C07276=1045.555,91.090,414.139,170.365,36.249,156.822
C07277=1045.549,90.841,414.159,170.363,36.248,156.822
C07278=1045.543,90.592,414.178,170.362,36.246,156.822
C07279=1045.537,90.343,414.197,170.359,36.245,156.821
C07280=1045.531,90.094,414.216,170.357,36.243,156.821
C07281=1045.524,89.845,414.234,170.356,36.242,156.821
C07282=1045.518,89.596,414.253,170.354,36.240,156.820
C07283=1045.512,89.345,414.272,170.352,36.239,156.820
C07284=1045.505,89.096,414.291,170.351,36.238,156.820
C07285=1045.499,88.847,414.310,170.349,36.236,156.820
C07286=1045.493,88.598,414.329,170.346,36.234,156.819
C07287=1045.487,88.349,414.348,170.345,36.233,156.819
C07288=1045.480,88.099,414.366,170.343,36.232,156.819
C07289=1045.474,87.850,414.385,170.341,36.231,156.819
C07290=1045.467,87.601,414.404,170.340,36.229,156.818
C07291=1045.462,87.352,414.423,170.338,36.228,156.818
C07292=1045.455,87.103,414.441,170.335,36.226,156.818
C07293=1045.449,86.854,414.460,170.334,36.224,156.817
C07294=1045.442,86.604,414.479,170.332,36.223,156.817
C07295=1045.437,86.355,414.498,170.330,36.222,156.817
C07296=1045.430,86.106,414.517,170.329,36.221,156.817
C07297=1045.424,85.857,414.535,170.327,36.219,156.816
C07298=1045.418,85.608,414.554,170.325,36.217,156.816
C07299=1045.412,85.358,414.573,170.323,36.216,156.816
C07300=1045.405,85.109,414.592,170.321,36.214,156.816
C07301=1045.399,84.860,414.610,170.319,36.213,156.815
C07302=1045.393,84.611,414.629,170.318,36.212,156.815
C07303=1045.387,84.361,414.648,170.316,36.211,156.815
C07304=1045.380,84.112,414.667,170.314,36.209,156.815
C07305=1045.374,83.863,414.685,170.313,36.207,156.814
C07306=1045.368,83.614,414.703,170.310,36.206,156.814
C07307=1045.362,83.365,414.722,170.308,36.204,156.814
C07308=1045.356,83.116,414.741,170.307,36.203,156.813
C07309=1045.350,82.866,414.760,170.305,36.202,156.813
C07310=1045.344,82.617,414.778,170.303,36.200,156.813
C07311=1045.337,82.368,414.797,170.302,36.199,156.813
C07312=1045.331,82.118,414.815,170.300,36.197,156.812
C07313=1045.325,81.869,414.834,170.297,36.195,156.812
C07314=1045.319,81.620,414.853,170.296,36.194,156.812
C07315=1045.312,81.371,414.872,170.294,36.193,156.812
C07316=1045.306,81.122,414.890,170.292,36.192,156.811
C07317=1045.300,80.873,414.909,170.291,36.190,156.811
C07318=1045.295,80.623,414.927,170.289,36.188,156.811
C07319=1045.288,80.374,414.946,170.288,36.187,156.811
C07320=1045.282,80.125,414.964,170.285,36.185,156.810
C07321=1045.276,79.876,414.983,170.283,36.184,156.810
C07322=1045.269,79.626,415.001,170.282,36.183,156.810
C07323=1045.264,79.408,415.018,170.280,36.181,156.809
C07324=1045.259,79.189,415.034,170.279,36.180,156.809
C07325=1045.254,78.971,415.050,170.277,36.178,156.809
C07326=1045.248,78.752,415.066,170.275,36.177,156.809
C07327=1045.243,78.533,415.083,170.273,36.176,156.808
C07328=1045.237,78.314,415.099,170.272,36.175,156.808
C07329=1045.231,78.096,415.115,170.270,36.173,156.808
C07330=1045.227,77.877,415.131,170.269,36.172,156.808
C07331=1045.219,77.591,415.152,170.267,36.171,156.807
C07332=1045.212,77.306,415.173,170.265,36.169,156.807
C07333=1045.205,77.019,415.194,170.263,36.168,156.807
C07334=1045.198,76.733,415.215,170.260,36.166,156.807
C07335=1045.192,76.484,415.234,170.259,36.164,156.806
C07336=1045.185,76.235,415.252,170.257,36.163,156.806
C07337=1045.179,75.985,415.270,170.255,36.161,156.806
C07338=1045.173,75.736,415.289,170.254,36.160,156.805
C07339=1045.167,75.487,415.307,170.252,36.159,156.805
C07340=1045.160,75.237,415.325,170.250,36.158,156.805
C07341=1045.154,74.988,415.343,170.248,36.156,156.805
C07342=1045.148,74.739,415.362,170.246,36.154,156.804
C07343=1045.142,74.490,415.380,170.244,36.153,156.804
C07344=1045.135,74.241,415.398,170.243,36.152,156.804
C07345=1045.129,73.992,415.416,170.241,36.151,156.804
C07346=1045.122,73.742,415.434,170.239,36.149,156.803
C07347=1045.117,73.494,415.452,170.238,36.147,156.803
C07348=1045.111,73.244,415.470,170.235,36.146,156.803
C07349=1045.104,72.995,415.489,170.233,36.145,156.803
C07350=1045.098,72.745,415.507,170.232,36.143,156.802
C07351=1045.092,72.496,415.526,170.230,36.142,156.802
C07352=1045.085,72.246,415.544,170.228,36.140,156.802
C07353=1045.080,71.998,415.562,170.227,36.139,156.802
C07354=1045.073,71.748,415.580,170.225,36.137,156.801
C07355=1045.067,71.499,415.598,170.222,36.136,156.801
C07356=1045.060,71.249,415.616,170.221,36.135,156.801
C07357=1045.054,71.001,415.634,170.219,36.134,156.801
C07358=1045.048,70.751,415.652,170.217,36.132,156.800
C07359=1045.042,70.502,415.671,170.216,36.130,156.800
C07360=1045.036,70.252,415.689,170.214,36.129,156.800
C07361=1045.030,70.003,415.706,170.213,36.128,156.800
C07362=1045.024,69.754,415.725,170.210,36.126,156.799
C07363=1045.018,69.504,415.743,170.208,36.125,156.799
C07364=1045.010,69.256,415.761,170.207,36.123,156.799
C07365=1045.004,69.006,415.779,170.205,36.122,156.799
C07366=1044.999,68.757,415.796,170.203,36.121,156.798
C07367=1044.992,68.508,415.815,170.202,36.119,156.798
C07368=1044.986,68.258,415.832,170.200,36.118,156.798
C07369=1044.979,68.009,415.850,170.197,36.116,156.797
C07370=1044.974,67.760,415.868,170.196,36.115,156.797
C07371=1044.967,67.510,415.886,170.194,36.114,156.797
C07372=1044.961,67.261,415.904,170.192,36.112,156.797
C07373=1044.954,67.012,415.922,170.191,36.111,156.796
C07374=1044.949,66.763,415.940,170.189,36.109,156.796
C07375=1044.943,66.513,415.958,170.187,36.108,156.796
C07376=1044.935,66.264,415.976,170.186,36.107,156.796
C07377=1044.930,66.015,415.994,170.183,36.106,156.795
C07378=1044.924,65.765,416.011,170.181,36.104,156.795
C07379=1044.917,65.516,416.029,170.180,36.102,156.795
C07380=1044.910,65.267,416.047,170.178,36.101,156.795
C07381=1044.905,65.018,416.065,170.176,36.100,156.794
C07382=1044.898,64.768,416.082,170.174,36.099,156.794
C07383=1044.892,64.519,416.100,170.173,36.097,156.794
C07384=1044.886,64.270,416.119,170.170,36.095,156.794
C07385=1044.880,64.020,416.136,170.168,36.094,156.793
C07386=1044.873,63.771,416.154,170.167,36.093,156.793
C07387=1044.866,63.522,416.171,170.165,36.092,156.793
C07388=1044.861,63.273,416.189,170.163,36.090,156.793
C07389=1044.854,63.023,416.206,170.162,36.089,156.792
C07390=1044.848,62.773,416.224,170.160,36.088,156.792
C07391=1044.841,62.525,416.242,170.158,36.087,156.792
C07392=1044.835,62.276,416.260,170.156,36.085,156.792
C07393=1044.828,62.026,416.277,170.154,36.084,156.792
C07394=1044.822,61.776,416.295,170.152,36.083,156.791
C07395=1044.814,61.491,416.314,170.150,36.081,156.791
C07396=1044.807,61.204,416.335,170.148,36.080,156.791
C07397=1044.800,60.918,416.355,170.146,36.078,156.791
C07398=1044.792,60.632,416.375,170.144,36.076,156.790
C07399=1044.787,60.383,416.392,170.142,36.075,156.790
C07400=1044.780,60.133,416.410,170.140,36.074,156.790
C07401=1044.773,59.884,416.427,170.138,36.073,156.789
C07402=1044.768,59.635,416.445,170.137,36.071,156.789
C07403=1044.760,59.386,416.463,170.135,36.070,156.789
C07404=1044.754,59.136,416.481,170.133,36.069,156.789
C07405=1044.748,58.887,416.498,170.132,36.067,156.789
C07406=1044.742,58.638,416.516,170.130,36.066,156.788
C07407=1044.735,58.388,416.533,170.128,36.065,156.788
C07408=1044.729,58.139,416.550,170.126,36.063,156.788
C07409=1044.723,57.890,416.568,170.124,36.062,156.788
C07410=1044.716,57.641,416.585,170.122,36.060,156.787
C07411=1044.711,57.391,416.602,170.120,36.059,156.787
C07412=1044.704,57.141,416.619,170.119,36.058,156.787
C07413=1044.698,56.892,416.636,170.117,36.057,156.787
C07414=1044.691,56.643,416.654,170.115,36.055,156.786
C07415=1044.685,56.393,416.672,170.113,36.054,156.786
C07416=1044.679,56.144,416.689,170.111,36.053,156.786
C07417=1044.672,55.895,416.706,170.109,36.052,156.786
C07418=1044.666,55.646,416.723,170.108,36.050,156.785
C07419=1044.660,55.396,416.741,170.106,36.048,156.785
C07420=1044.653,55.147,416.759,170.104,36.047,156.785
C07421=1044.647,54.898,416.776,170.103,36.046,156.785
C07422=1044.641,54.648,416.794,170.101,36.045,156.784
C07423=1044.634,54.400,416.811,170.098,36.043,156.784
C07424=1044.628,54.149,416.828,170.097,36.042,156.784
C07425=1044.622,53.901,416.845,170.095,36.041,156.784
C07426=1044.615,53.651,416.862,170.093,36.039,156.783
C07427=1044.610,53.402,416.880,170.091,36.038,156.783
C07428=1044.603,53.153,416.897,170.090,36.037,156.783
C07429=1044.596,52.903,416.914,170.088,36.035,156.783
C07430=1044.591,52.654,416.932,170.086,36.034,156.782
C07431=1044.584,52.404,416.949,170.084,36.032,156.782
C07432=1044.579,52.155,416.966,170.082,36.031,156.782
C07433=1044.572,51.906,416.983,170.080,36.030,156.782
C07434=1044.565,51.657,417.000,170.079,36.029,156.782
C07435=1044.559,51.407,417.018,170.077,36.027,156.781
C07436=1044.553,51.158,417.035,170.075,36.026,156.781
C07437=1044.546,50.908,417.052,170.074,36.024,156.781
C07438=1044.541,50.659,417.070,170.072,36.023,156.780
C07439=1044.534,50.410,417.087,170.069,36.022,156.780
C07440=1044.528,50.161,417.103,170.068,36.020,156.780
C07441=1044.522,49.911,417.121,170.066,36.019,156.780
C07442=1044.516,49.662,417.138,170.064,36.018,156.780
C07443=1044.509,49.413,417.155,170.063,36.016,156.779
C07444=1044.504,49.163,417.172,170.061,36.015,156.779
C07445=1044.497,48.914,417.190,170.059,36.013,156.779
C07446=1044.491,48.665,417.207,170.057,36.012,156.779
C07447=1044.485,48.416,417.224,170.055,36.011,156.778
C07448=1044.479,48.166,417.241,170.053,36.009,156.778
C07449=1044.472,47.917,417.258,170.051,36.008,156.778
C07450=1044.466,47.667,417.276,170.050,36.007,156.778
C07451=1044.460,47.418,417.292,170.048,36.006,156.777
C07452=1044.453,47.169,417.309,170.046,36.004,156.777
C07453=1044.448,46.920,417.327,170.045,36.002,156.777
C07454=1044.441,46.670,417.343,170.043,36.001,156.777
C07455=1044.435,46.421,417.360,170.040,36.000,156.776
C07456=1044.429,46.172,417.378,170.039,35.999,156.776
C07457=1044.423,45.922,417.395,170.037,35.997,156.776
C07458=1044.417,45.673,417.412,170.035,35.996,156.776
C07459=1044.410,45.386,417.431,170.033,35.994,156.775
C07460=1044.402,45.100,417.451,170.031,35.993,156.775
C07461=1044.396,44.813,417.470,170.029,35.991,156.775
C07462=1044.389,44.527,417.490,170.027,35.990,156.775
C07463=1044.382,44.277,417.507,170.025,35.988,156.774
C07464=1044.376,44.029,417.524,170.023,35.986,156.774
C07465=1044.371,43.779,417.541,170.021,35.985,156.774
C07466=1044.364,43.529,417.558,170.020,35.984,156.774
C07467=1044.358,43.280,417.574,170.018,35.983,156.773
C07468=1044.351,43.031,417.592,170.016,35.981,156.773
C07469=1044.345,42.781,417.608,170.015,35.980,156.773
C07470=1044.340,42.532,417.625,170.013,35.979,156.773
C07471=1044.333,42.282,417.642,170.010,35.977,156.772
C07472=1044.327,42.033,417.659,170.009,35.976,156.772
C07473=1044.320,41.783,417.676,170.007,35.975,156.772
C07474=1044.314,41.535,417.693,170.005,35.974,156.772
C07475=1044.308,41.285,417.709,170.003,35.972,156.771
C07476=1044.301,41.036,417.726,170.002,35.971,156.771
C07477=1044.295,40.787,417.743,170.000,35.970,156.771
C07478=1044.289,40.536,417.759,169.998,35.968,156.771
C07479=1044.283,40.288,417.776,169.996,35.967,156.770
C07480=1044.277,40.038,417.792,169.994,35.965,156.770
C07481=1044.270,39.789,417.810,169.992,35.964,156.770
C07482=1044.264,39.540,417.826,169.990,35.963,156.770
C07483=1044.258,39.290,417.842,169.989,35.961,156.770
C07484=1044.251,39.041,417.860,169.987,35.960,156.769
C07485=1044.245,38.792,417.876,169.985,35.959,156.769
C07486=1044.239,38.543,417.893,169.984,35.958,156.769
C07487=1044.232,38.293,417.909,169.981,35.956,156.769
C07488=1044.227,38.043,417.926,169.979,35.955,156.768
C07489=1044.221,37.794,417.943,169.977,35.954,156.768
C07490=1044.214,37.544,417.960,169.976,35.952,156.768
C07491=1044.207,37.295,417.976,169.974,35.951,156.768
C07492=1044.202,37.046,417.992,169.972,35.950,156.767
C07493=1044.195,36.796,418.009,169.970,35.949,156.767
C07494=1044.189,36.547,418.025,169.969,35.947,156.767
C07495=1044.183,36.298,418.042,169.967,35.946,156.767
C07496=1044.176,36.048,418.059,169.964,35.945,156.767
C07497=1044.170,35.799,418.075,169.962,35.943,156.766
C07498=1044.163,35.550,418.091,169.961,35.942,156.766
C07499=1044.157,35.300,418.107,169.959,35.942,156.766
C07500=1044.151,35.051,418.124,169.957,35.940,156.766
C07501=1044.144,34.802,418.141,169.956,35.939,156.766
C07502=1044.138,34.552,418.157,169.954,35.938,156.765
C07503=1044.132,34.302,418.174,169.952,35.936,156.765
C07504=1044.125,34.053,418.189,169.950,35.935,156.765
C07505=1044.119,33.803,418.206,169.948,35.934,156.765
C07506=1044.112,33.555,418.223,169.946,35.933,156.764
C07507=1044.107,33.305,418.239,169.944,35.931,156.764
C07508=1044.101,33.056,418.255,169.942,35.930,156.764
C07509=1044.093,32.806,418.271,169.941,35.929,156.764
C07510=1044.087,32.557,418.288,169.939,35.927,156.763
C07511=1044.081,32.308,418.304,169.937,35.926,156.763
C07512=1044.075,32.059,418.321,169.935,35.925,156.763
C07513=1044.069,31.809,418.338,169.934,35.924,156.763
C07514=1044.062,31.560,418.353,169.931,35.922,156.763
C07515=1044.056,31.310,418.369,169.929,35.921,156.762
C07516=1044.050,31.061,418.386,169.927,35.920,156.762
C07517=1044.043,30.811,418.402,169.926,35.918,156.762
C07518=1044.037,30.562,418.419,169.924,35.917,156.762
C07519=1044.031,30.313,418.434,169.922,35.916,156.761
C07520=1044.025,30.063,418.450,169.920,35.914,156.761
C07521=1044.018,29.813,418.467,169.919,35.914,156.761
C07522=1044.012,29.564,418.484,169.917,35.913,156.761
C07523=1044.005,29.278,418.502,169.914,35.911,156.761
C07524=1043.998,28.991,418.521,169.912,35.909,156.760
C07525=1043.991,28.705,418.540,169.910,35.908,156.760
C07526=1043.984,28.418,418.558,169.908,35.907,156.760
C07527=1043.978,28.169,418.574,169.906,35.905,156.760
C07528=1043.971,27.919,418.590,169.904,35.904,156.759
C07529=1043.965,27.669,418.606,169.903,35.903,156.759
C07530=1043.958,27.420,418.622,169.901,35.902,156.759
C07531=1043.952,27.171,418.638,169.899,35.900,156.759
C07532=1043.946,26.922,418.655,169.896,35.899,156.759
C07533=1043.939,26.672,418.671,169.895,35.898,156.758
C07534=1043.933,26.423,418.687,169.893,35.896,156.758
C07535=1043.927,26.173,418.703,169.891,35.896,156.758
C07536=1043.920,25.924,418.719,169.889,35.894,156.758
C07537=1043.914,25.675,418.735,169.887,35.893,156.757
C07538=1043.907,25.425,418.751,169.886,35.892,156.757
C07539=1043.901,25.176,418.767,169.884,35.891,156.757
C07540=1043.894,24.927,418.783,169.882,35.889,156.757
C07541=1043.889,24.677,418.798,169.879,35.888,156.757
C07542=1043.883,24.427,418.815,169.878,35.887,156.756
C07543=1043.876,24.178,418.830,169.876,35.886,156.756
C07544=1043.869,23.928,418.847,169.874,35.885,156.756
C07545=1043.863,23.679,418.863,169.872,35.883,156.756
C07546=1043.857,23.430,418.879,169.870,35.882,156.756
C07547=1043.850,23.181,418.895,169.869,35.881,156.755
C07548=1043.844,22.931,418.910,169.867,35.880,156.755
C07549=1043.839,22.682,418.926,169.865,35.879,156.755
C07550=1043.832,22.433,418.942,169.863,35.878,156.755
C07551=1043.825,22.183,418.959,169.861,35.876,156.755
C07552=1043.819,21.934,418.974,169.859,35.875,156.754
C07553=1043.813,21.684,418.990,169.857,35.874,156.754
C07554=1043.806,21.434,419.006,169.855,35.872,156.754
C07555=1043.800,21.185,419.022,169.853,35.871,156.754
C07556=1043.794,20.936,419.037,169.852,35.870,156.753
C07557=1043.788,20.686,419.053,169.850,35.869,156.753
C07558=1043.781,20.437,419.069,169.848,35.868,156.753
C07559=1043.775,20.188,419.085,169.846,35.867,156.753
C07560=1043.769,19.938,419.101,169.844,35.865,156.753
C07561=1043.762,19.688,419.116,169.842,35.864,156.752
C07562=1043.756,19.439,419.132,169.840,35.863,156.752
C07563=1043.750,19.190,419.148,169.838,35.861,156.752
C07564=1043.743,18.940,419.163,169.836,35.861,156.752
C07565=1043.737,18.691,419.180,169.834,35.859,156.752
C07566=1043.731,18.442,419.195,169.833,35.858,156.751
C07567=1043.724,18.192,419.210,169.831,35.857,156.751
C07568=1043.718,17.943,419.226,169.829,35.856,156.751
C07569=1043.712,17.694,419.242,169.827,35.855,156.751
C07570=1043.706,17.444,419.258,169.825,35.854,156.751
C07571=1043.699,17.195,419.273,169.823,35.852,156.750
C07572=1043.693,16.946,419.289,169.821,35.851,156.750
C07573=1043.687,16.696,419.305,169.819,35.850,156.750
C07574=1043.680,16.447,419.320,169.817,35.849,156.750
C07575=1043.675,16.197,419.336,169.815,35.848,156.750
C07576=1043.668,15.948,419.351,169.814,35.847,156.749
C07577=1043.661,15.698,419.367,169.812,35.845,156.749
C07578=1043.655,15.448,419.383,169.810,35.844,156.749
C07579=1043.648,15.199,419.399,169.808,35.843,156.749
C07580=1043.643,14.949,419.414,169.806,35.842,156.749
C07581=1043.636,14.700,419.430,169.804,35.841,156.748
C07582=1043.630,14.450,419.445,169.802,35.839,156.748
C07583=1043.624,14.201,419.461,169.800,35.838,156.748
C07584=1043.617,13.951,419.476,169.798,35.837,156.748
C07585=1043.611,13.702,419.492,169.796,35.836,156.748
C07586=1043.604,13.452,419.507,169.794,35.835,156.747
C07587=1043.597,13.167,419.524,169.792,35.834,156.747
C07588=1043.589,12.882,419.542,169.790,35.832,156.747
C07589=1043.582,12.597,419.559,169.788,35.831,156.747
C07590=1043.575,12.312,419.578,169.786,35.830,156.747
C07591=1043.569,12.062,419.592,169.784,35.829,156.746
C07592=1043.562,11.813,419.608,169.781,35.828,156.746
C07593=1043.556,11.564,419.623,169.779,35.827,156.746
C07594=1043.550,11.314,419.638,169.778,35.826,156.746
C07595=1043.543,11.065,419.654,169.776,35.824,156.746
C07596=1043.537,10.815,419.669,169.774,35.823,156.745
C07597=1043.531,10.566,419.685,169.772,35.822,156.745
C07598=1043.524,10.316,419.700,169.770,35.821,156.745
C07599=1043.518,10.067,419.715,169.768,35.820,156.745
C07600=1043.511,9.818,419.730,169.766,35.819,156.745
C07601=1043.505,9.568,419.745,169.765,35.818,156.745
C07602=1043.498,9.318,419.760,169.762,35.817,156.744
C07603=1043.492,9.069,419.776,169.760,35.816,156.744
C07604=1043.485,8.820,419.791,169.758,35.815,156.744
C07605=1043.480,8.570,419.806,169.756,35.813,156.744
C07606=1043.473,8.321,419.822,169.754,35.813,156.744
C07607=1043.467,8.071,419.837,169.752,35.811,156.743
C07608=1043.460,7.821,419.852,169.751,35.810,156.743
C07609=1043.453,7.572,419.868,169.749,35.809,156.743
C07610=1043.447,7.323,419.883,169.747,35.808,156.743
C07611=1043.441,7.073,419.898,169.745,35.807,156.743
C07612=1043.435,6.824,419.912,169.743,35.806,156.743
C07613=1043.428,6.575,419.928,169.741,35.805,156.742
C07614=1043.422,6.325,419.943,169.738,35.803,156.742
C07615=1043.416,6.075,419.958,169.737,35.803,156.742
C07616=1043.410,5.826,419.973,169.735,35.801,156.742
C07617=1043.403,5.577,419.989,169.733,35.800,156.742
C07618=1043.397,5.327,420.004,169.731,35.799,156.741
C07619=1043.390,5.077,420.019,169.729,35.798,156.741
C07620=1043.384,4.828,420.034,169.727,35.797,156.741
C07621=1043.378,4.579,420.048,169.725,35.796,156.741
C07622=1043.372,4.330,420.064,169.724,35.795,156.741
C07623=1043.365,4.080,420.079,169.722,35.794,156.740
C07624=1043.359,3.830,420.094,169.720,35.792,156.740
C07625=1043.352,3.581,420.109,169.717,35.792,156.740
C07626=1043.347,3.331,420.124,169.715,35.790,156.740
C07627=1043.340,3.081,420.139,169.713,35.789,156.740
C07628=1043.334,2.833,420.155,169.711,35.788,156.740
C07629=1043.328,2.583,420.170,169.709,35.787,156.739
C07630=1043.322,2.333,420.185,169.708,35.786,156.739
C07631=1043.315,2.084,420.199,169.706,35.785,156.739
C07632=1043.309,1.834,420.214,169.704,35.784,156.739
C07633=1043.303,1.585,420.229,169.702,35.783,156.739
C07634=1043.297,1.335,420.244,169.700,35.781,156.738
C07635=1043.290,1.086,420.259,169.698,35.781,156.738
C07636=1043.284,0.837,420.275,169.695,35.779,156.738
C07637=1043.277,0.587,420.290,169.693,35.778,156.738
C07638=1043.271,0.338,420.304,169.692,35.777,156.738
C07639=1043.265,0.088,420.319,169.690,35.776,156.737
C07640=1043.259,-0.161,420.334,169.688,35.775,156.737
C07641=1043.252,-0.411,420.349,169.686,35.774,156.737
C07642=1043.246,-0.661,420.364,169.684,35.773,156.737
C07643=1043.241,-0.910,420.379,169.682,35.771,156.737
C07644=1043.234,-1.159,420.394,169.680,35.771,156.737
C07645=1043.228,-1.409,420.409,169.678,35.769,156.736
C07646=1043.222,-1.659,420.424,169.677,35.768,156.736
C07647=1043.216,-1.908,420.438,169.675,35.767,156.736
C07648=1043.209,-2.157,420.453,169.672,35.766,156.736
C07649=1043.203,-2.407,420.468,169.670,35.765,156.736
C07650=1043.197,-2.656,420.483,169.668,35.763,156.735
C07651=1043.190,-2.939,420.499,169.666,35.762,156.735
C07652=1043.182,-3.223,420.517,169.664,35.762,156.735
C07653=1043.176,-3.507,420.534,169.662,35.760,156.735
C07654=1043.169,-3.790,420.550,169.659,35.759,156.735
C07655=1043.162,-4.040,420.564,169.657,35.758,156.734
C07656=1043.156,-4.289,420.579,169.655,35.757,156.734
C07657=1043.150,-4.538,420.594,169.654,35.756,156.734
C07658=1043.143,-4.788,420.609,169.652,35.755,156.734
C07659=1043.136,-5.037,420.623,169.649,35.754,156.734
C07660=1043.130,-5.286,420.638,169.647,35.753,156.734
C07661=1043.124,-5.536,420.652,169.645,35.752,156.733
C07662=1043.118,-5.786,420.667,169.643,35.751,156.733
C07663=1043.111,-6.035,420.681,169.641,35.750,156.733
C07664=1043.105,-6.284,420.696,169.639,35.749,156.733
C07665=1043.098,-6.534,420.711,169.637,35.748,156.733
C07666=1043.092,-6.784,420.724,169.635,35.747,156.733
C07667=1043.086,-7.033,420.739,169.633,35.746,156.732
C07668=1043.080,-7.283,420.754,169.631,35.745,156.732
C07669=1043.073,-7.532,420.769,169.629,35.744,156.732
C07670=1043.066,-7.782,420.783,169.627,35.743,156.732
C07671=1043.061,-8.031,420.797,169.625,35.742,156.732
C07672=1043.054,-8.281,420.812,169.623,35.741,156.732
C07673=1043.047,-8.530,420.826,169.620,35.740,156.731
C07674=1043.042,-8.780,420.840,169.619,35.739,156.731
C07675=1043.035,-9.029,420.855,169.617,35.738,156.731
C07676=1043.028,-9.279,420.870,169.615,35.737,156.731
C07677=1043.022,-9.528,420.884,169.613,35.736,156.731
C07678=1043.016,-9.778,420.898,169.611,35.735,156.731
C07679=1043.010,-10.028,420.913,169.609,35.734,156.730
C07680=1043.003,-10.276,420.927,169.607,35.733,156.730
C07681=1042.997,-10.527,420.942,169.605,35.732,156.730
C07682=1042.991,-10.776,420.956,169.603,35.731,156.730
C07683=1042.984,-11.025,420.971,169.601,35.730,156.730
C07684=1042.978,-11.275,420.985,169.599,35.729,156.730
C07685=1042.972,-11.524,420.999,169.597,35.728,156.729
C07686=1042.965,-11.774,421.014,169.594,35.727,156.729
C07687=1042.959,-12.024,421.028,169.592,35.726,156.729
C07688=1042.953,-12.273,421.042,169.590,35.725,156.729
C07689=1042.947,-12.523,421.056,169.588,35.724,156.729
C07690=1042.941,-12.772,421.071,169.586,35.723,156.729
C07691=1042.934,-13.021,421.086,169.584,35.722,156.728
C07692=1042.928,-13.271,421.099,169.582,35.721,156.728
C07693=1042.922,-13.520,421.114,169.580,35.720,156.728
C07694=1042.916,-13.771,421.128,169.578,35.719,156.728
C07695=1042.909,-14.019,421.142,169.576,35.718,156.728
C07696=1042.903,-14.269,421.157,169.574,35.717,156.728
C07697=1042.897,-14.518,421.171,169.573,35.716,156.728
C07698=1042.890,-14.768,421.185,169.571,35.715,156.727
C07699=1042.885,-15.017,421.199,169.568,35.714,156.727
C07700=1042.878,-15.267,421.214,169.566,35.713,156.727
C07701=1042.872,-15.517,421.228,169.564,35.713,156.727
C07702=1042.865,-15.766,421.242,169.562,35.711,156.727
C07703=1042.859,-16.016,421.256,169.560,35.711,156.727
C07704=1042.853,-16.264,421.270,169.558,35.710,156.727
C07705=1042.846,-16.515,421.284,169.556,35.709,156.726
C07706=1042.840,-16.765,421.298,169.554,35.708,156.726
C07707=1042.834,-17.014,421.312,169.552,35.707,156.726
C07708=1042.827,-17.264,421.326,169.550,35.706,156.726
C07709=1042.820,-17.512,421.340,169.548,35.705,156.726
C07710=1042.814,-17.763,421.354,169.546,35.704,156.726
C07711=1042.808,-18.012,421.367,169.544,35.703,156.725
C07712=1042.802,-18.262,421.382,169.542,35.702,156.725
C07713=1042.796,-18.511,421.396,169.540,35.702,156.725
C07714=1042.789,-18.760,421.411,169.537,35.700,156.725
C07715=1042.782,-19.043,421.426,169.534,35.700,156.725
C07716=1042.775,-19.324,421.442,169.532,35.698,156.725
C07717=1042.768,-19.606,421.458,169.530,35.698,156.725
C07718=1042.761,-19.888,421.473,169.527,35.696,156.724
C07719=1042.754,-20.137,421.487,169.525,35.696,156.724
C07720=1042.748,-20.386,421.501,169.523,35.694,156.724
C07721=1042.742,-20.636,421.515,169.521,35.694,156.724
C07722=1042.735,-20.885,421.529,169.519,35.693,156.724
C07723=1042.729,-21.135,421.543,169.517,35.692,156.724
C07724=1042.723,-21.385,421.556,169.515,35.691,156.724
C07725=1042.717,-21.635,421.570,169.513,35.690,156.723
C07726=1042.710,-21.884,421.584,169.511,35.689,156.723
C07727=1042.703,-22.133,421.598,169.509,35.688,156.723
C07728=1042.698,-22.383,421.612,169.507,35.688,156.723
C07729=1042.691,-22.633,421.626,169.504,35.686,156.723
C07730=1042.684,-22.882,421.640,169.502,35.686,156.723
C07731=1042.678,-23.132,421.654,169.500,35.685,156.723
C07732=1042.672,-23.381,421.667,169.498,35.684,156.722
C07733=1042.667,-23.631,421.681,169.496,35.683,156.722
C07734=1042.660,-23.880,421.695,169.494,35.682,156.722
C07735=1042.653,-24.129,421.709,169.492,35.681,156.722
C07736=1042.647,-24.380,421.723,169.490,35.680,156.722
C07737=1042.641,-24.629,421.736,169.488,35.680,156.722
C07738=1042.635,-24.878,421.749,169.486,35.679,156.722
C07739=1042.628,-25.128,421.764,169.484,35.678,156.721
C07740=1042.622,-25.377,421.778,169.482,35.677,156.721
C07741=1042.615,-25.627,421.791,169.480,35.676,156.721
C07742=1042.610,-25.877,421.805,169.478,35.675,156.721
C07743=1042.604,-26.126,421.818,169.476,35.674,156.721
C07744=1042.598,-26.376,421.833,169.474,35.674,156.721
C07745=1042.591,-26.625,421.846,169.471,35.672,156.721
C07746=1042.585,-26.874,421.860,169.469,35.672,156.720
C07747=1042.578,-27.124,421.873,169.467,35.671,156.720
C07748=1042.573,-27.374,421.887,169.464,35.670,156.720
C07749=1042.566,-27.624,421.901,169.462,35.669,156.720
C07750=1042.560,-27.873,421.914,169.460,35.668,156.720
C07751=1042.553,-28.122,421.927,169.458,35.668,156.720
C07752=1042.547,-28.372,421.941,169.456,35.667,156.720
C07753=1042.540,-28.621,421.954,169.454,35.666,156.720
C07754=1042.534,-28.871,421.968,169.452,35.666,156.720
C07755=1042.527,-29.121,421.981,169.450,35.664,156.719
C07756=1042.522,-29.370,421.995,169.448,35.664,156.719
C07757=1042.515,-29.620,422.009,169.446,35.663,156.719
C07758=1042.509,-29.869,422.022,169.444,35.662,156.719
C07759=1042.503,-30.119,422.035,169.442,35.661,156.719
C07760=1042.496,-30.369,422.049,169.440,35.661,156.719
C07761=1042.490,-30.618,422.062,169.437,35.659,156.719
C07762=1042.483,-30.867,422.075,169.435,35.659,156.718
C07763=1042.477,-31.117,422.089,169.432,35.658,156.718
C07764=1042.470,-31.366,422.102,169.430,35.657,156.718
C07765=1042.464,-31.616,422.115,169.428,35.657,156.718
C07766=1042.458,-31.867,422.129,169.426,35.656,156.718
C07767=1042.452,-32.116,422.142,169.424,35.655,156.718
C07768=1042.446,-32.365,422.156,169.422,35.654,156.718
C07769=1042.439,-32.615,422.169,169.420,35.653,156.718
C07770=1042.433,-32.864,422.183,169.418,35.653,156.718
C07771=1042.427,-33.114,422.196,169.416,35.652,156.717
C07772=1042.420,-33.363,422.209,169.413,35.651,156.717
C07773=1042.414,-33.613,422.223,169.411,35.651,156.717
C07774=1042.408,-33.863,422.235,169.409,35.650,156.717
C07775=1042.402,-34.112,422.249,169.407,35.649,156.717
C07776=1042.395,-34.361,422.262,169.405,35.648,156.717
C07777=1042.389,-34.611,422.276,169.403,35.647,156.717
C07778=1042.382,-34.860,422.289,169.401,35.647,156.717
C07779=1042.376,-35.142,422.304,169.398,35.646,156.716
C07780=1042.369,-35.422,422.319,169.396,35.644,156.716
C07781=1042.362,-35.704,422.334,169.394,35.644,156.716
C07782=1042.354,-35.985,422.349,169.390,35.643,156.716
C07783=1042.348,-36.234,422.362,169.388,35.642,156.716
C07784=1042.342,-36.484,422.375,169.386,35.642,156.716
C07785=1042.336,-36.733,422.388,169.384,35.641,156.716
C07786=1042.330,-36.982,422.401,169.382,35.640,156.716
C07787=1042.323,-37.232,422.415,169.380,35.639,156.715
C07788=1042.317,-37.482,422.427,169.378,35.638,156.715
C07789=1042.311,-37.732,422.441,169.376,35.638,156.715
C07790=1042.305,-37.981,422.454,169.373,35.637,156.715
C07791=1042.299,-38.231,422.466,169.371,35.636,156.715
C07792=1042.292,-38.481,422.480,169.369,35.636,156.715
C07793=1042.286,-38.730,422.493,169.367,35.635,156.715
C07794=1042.280,-38.980,422.506,169.365,35.634,156.715
C07795=1042.274,-39.229,422.519,169.363,35.634,156.715
C07796=1042.267,-39.478,422.532,169.361,35.633,156.715
C07797=1042.261,-39.729,422.545,169.358,35.632,156.714
C07798=1042.255,-39.978,422.559,169.356,35.631,156.714
C07799=1042.248,-40.227,422.571,169.354,35.631,156.714
C07800=1042.242,-40.477,422.584,169.352,35.630,156.714
C07801=1042.236,-40.726,422.597,169.350,35.629,156.714
C07802=1042.229,-40.977,422.610,169.348,35.629,156.714
C07803=1042.223,-41.226,422.623,169.345,35.628,156.714
C07804=1042.216,-41.476,422.635,169.342,35.627,156.714
C07805=1042.210,-41.725,422.648,169.340,35.627,156.714
C07806=1042.204,-41.974,422.662,169.338,35.626,156.714
C07807=1042.198,-42.224,422.674,169.336,35.625,156.713
C07808=1042.192,-42.473,422.688,169.334,35.625,156.713
C07809=1042.184,-42.724,422.700,169.332,35.624,156.713
C07810=1042.178,-42.973,422.713,169.329,35.623,156.713
C07811=1042.172,-43.223,422.726,169.327,35.622,156.713
C07812=1042.166,-43.472,422.739,169.325,35.622,156.713
C07813=1042.160,-43.722,422.752,169.323,35.621,156.713
C07814=1042.153,-43.971,422.764,169.321,35.621,156.713
C07815=1042.147,-44.221,422.777,169.319,35.620,156.713
C07816=1042.141,-44.470,422.790,169.316,35.620,156.713
C07817=1042.135,-44.720,422.803,169.314,35.619,156.713
C07818=1042.128,-44.970,422.816,169.312,35.618,156.712
C07819=1042.122,-45.219,422.828,169.310,35.618,156.712
C07820=1042.116,-45.469,422.841,169.308,35.617,156.712
C07821=1042.110,-45.719,422.854,169.306,35.616,156.712
C07822=1042.104,-45.969,422.867,169.303,35.615,156.712
C07823=1042.097,-46.217,422.879,169.301,35.615,156.712
C07824=1042.091,-46.467,422.892,169.299,35.614,156.712
C07825=1042.085,-46.717,422.904,169.297,35.613,156.712
C07826=1042.079,-46.967,422.918,169.295,35.613,156.712
C07827=1042.072,-47.216,422.930,169.291,35.612,156.711
C07828=1042.066,-47.465,422.943,169.290,35.612,156.712
C07829=1042.060,-47.715,422.955,169.287,35.611,156.711
C07830=1042.054,-47.965,422.968,169.285,35.611,156.711
C07831=1042.047,-48.214,422.981,169.283,35.610,156.711
C07832=1042.041,-48.464,422.993,169.281,35.609,156.711
C07833=1042.035,-48.714,423.006,169.278,35.609,156.711
C07834=1042.029,-48.963,423.019,169.276,35.608,156.711
C07835=1042.022,-49.213,423.031,169.274,35.607,156.711
C07836=1042.016,-49.463,423.044,169.272,35.606,156.711
C07837=1042.010,-49.712,423.057,169.270,35.606,156.711
C07838=1042.004,-49.961,423.069,169.267,35.605,156.710
C07839=1041.998,-50.211,423.081,169.265,35.605,156.711
C07840=1041.992,-50.461,423.094,169.263,35.604,156.710
C07841=1041.985,-50.710,423.107,169.261,35.604,156.710
C07842=1041.979,-50.960,423.119,169.259,35.603,156.710
C07843=1041.972,-51.242,423.133,169.256,35.603,156.710
C07844=1041.964,-51.523,423.147,169.254,35.602,156.710
C07845=1041.957,-51.805,423.160,169.251,35.601,156.710
C07846=1041.950,-52.086,423.174,169.248,35.601,156.710
C07847=1041.943,-52.335,423.186,169.246,35.601,156.710
C07848=1041.937,-52.585,423.199,169.244,35.600,156.710
C07849=1041.931,-52.835,423.211,169.242,35.599,156.710
C07850=1041.925,-53.084,423.224,169.239,35.599,156.710
C07851=1041.918,-53.334,423.236,169.237,35.599,156.710
C07852=1041.911,-53.583,423.248,169.235,35.598,156.710
C07853=1041.905,-53.833,423.261,169.233,35.598,156.710
C07854=1041.899,-54.083,423.273,169.230,35.597,156.709
C07855=1041.892,-54.332,423.285,169.228,35.596,156.709
C07856=1041.886,-54.582,423.297,169.226,35.596,156.709
C07857=1041.880,-54.832,423.309,169.224,35.596,156.709
C07858=1041.874,-55.082,423.322,169.221,35.596,156.709
C07859=1041.867,-55.331,423.334,169.219,35.595,156.709
C07860=1041.860,-55.581,423.346,169.216,35.594,156.709
C07861=1041.854,-55.831,423.358,169.214,35.594,156.709
C07862=1041.848,-56.080,423.370,169.211,35.593,156.709
C07863=1041.841,-56.330,423.382,169.209,35.593,156.709
C07864=1041.835,-56.580,423.395,169.207,35.593,156.709
C07865=1041.829,-56.829,423.407,169.205,35.592,156.709
C07866=1041.823,-57.078,423.418,169.202,35.592,156.709
C07867=1041.817,-57.328,423.431,169.200,35.591,156.709
C07868=1041.810,-57.578,423.443,169.198,35.591,156.709
C07869=1041.804,-57.828,423.455,169.196,35.591,156.709
C07870=1041.797,-58.077,423.467,169.193,35.590,156.709
C07871=1041.791,-58.327,423.479,169.191,35.589,156.708
C07872=1041.785,-58.577,423.492,169.189,35.589,156.708
C07873=1041.778,-58.826,423.504,169.187,35.588,156.708
C07874=1041.772,-59.075,423.515,169.184,35.588,156.708
C07875=1041.766,-59.325,423.528,169.182,35.588,156.708
C07876=1041.760,-59.574,423.540,169.180,35.587,156.708
C07877=1041.753,-59.824,423.552,169.177,35.587,156.708
C07878=1041.747,-60.074,423.564,169.175,35.586,156.708
C07879=1041.740,-60.323,423.576,169.173,35.586,156.708
C07880=1041.734,-60.574,423.587,169.171,35.585,156.708
C07881=1041.729,-60.823,423.600,169.168,35.585,156.708
C07882=1041.722,-61.072,423.612,169.166,35.585,156.708
C07883=1041.715,-61.322,423.624,169.164,35.584,156.708
C07884=1041.710,-61.572,423.636,169.161,35.584,156.708
C07885=1041.703,-61.821,423.648,169.159,35.583,156.708
C07886=1041.697,-62.070,423.660,169.157,35.583,156.708
C07887=1041.691,-62.321,423.671,169.155,35.582,156.708
C07888=1041.685,-62.570,423.683,169.152,35.582,156.708
C07889=1041.678,-62.820,423.695,169.150,35.582,156.708
C07890=1041.671,-63.070,423.707,169.148,35.581,156.707
C07891=1041.666,-63.319,423.720,169.146,35.581,156.707
C07892=1041.660,-63.569,423.731,169.143,35.580,156.707
C07893=1041.653,-63.818,423.743,169.141,35.580,156.707
C07894=1041.647,-64.068,423.755,169.139,35.579,156.707
C07895=1041.641,-64.317,423.767,169.136,35.579,156.707
C07896=1041.635,-64.567,423.778,169.134,35.579,156.707
C07897=1041.628,-64.817,423.790,169.132,35.578,156.707
C07898=1041.622,-65.067,423.803,169.129,35.578,156.707
C07899=1041.616,-65.316,423.814,169.127,35.577,156.707
C07900=1041.610,-65.566,423.826,169.125,35.577,156.707
C07901=1041.604,-65.816,423.838,169.123,35.577,156.707
C07902=1041.598,-66.065,423.850,169.120,35.576,156.707
C07903=1041.592,-66.315,423.861,169.118,35.576,156.707
C07904=1041.585,-66.564,423.873,169.116,35.576,156.707
C07905=1041.580,-66.814,423.885,169.113,35.575,156.707
C07906=1041.573,-67.064,423.896,169.111,35.575,156.707
C07907=1041.566,-67.346,423.910,169.108,35.574,156.707
C07908=1041.559,-67.629,423.923,169.105,35.574,156.707
C07909=1041.552,-67.912,423.936,169.103,35.573,156.707
C07910=1041.545,-68.195,423.949,169.100,35.573,156.706
C07911=1041.539,-68.444,423.961,169.097,35.573,156.707
C07912=1041.533,-68.693,423.974,169.095,35.572,156.706
C07913=1041.527,-68.944,423.985,169.093,35.572,156.706
C07914=1041.520,-69.193,423.997,169.090,35.571,156.706
C07915=1041.515,-69.443,424.008,169.088,35.571,156.706
C07916=1041.509,-69.693,424.020,169.086,35.570,156.706
C07917=1041.502,-69.942,424.032,169.084,35.570,156.706
C07918=1041.496,-70.192,424.043,169.081,35.570,156.706
C07919=1041.490,-70.441,424.055,169.079,35.570,156.706
C07920=1041.485,-70.691,424.066,169.077,35.569,156.706
C07921=1041.478,-70.941,424.078,169.074,35.569,156.706
C07922=1041.472,-71.191,424.090,169.072,35.568,156.706
C07923=1041.466,-71.440,424.101,169.070,35.568,156.706
C07924=1041.460,-71.690,424.113,169.067,35.567,156.706
C07925=1041.454,-71.939,424.125,169.065,35.567,156.706
C07926=1041.448,-72.189,424.136,169.063,35.567,156.706
C07927=1041.441,-72.439,424.148,169.060,35.567,156.706
C07928=1041.435,-72.688,424.159,169.058,35.566,156.706
C07929=1041.429,-72.938,424.171,169.056,35.566,156.706
C07930=1041.424,-73.188,424.182,169.053,35.565,156.706
C07931=1041.417,-73.437,424.194,169.051,35.565,156.706
C07932=1041.411,-73.687,424.205,169.049,35.564,156.706
C07933=1041.406,-73.937,424.217,169.046,35.564,156.706
C07934=1041.400,-74.186,424.228,169.044,35.564,156.706
C07935=1041.393,-74.436,424.240,169.042,35.564,156.705
C07936=1041.386,-74.685,424.251,169.039,35.563,156.705
C07937=1041.380,-74.935,424.262,169.037,35.563,156.706
C07938=1041.374,-75.185,424.273,169.035,35.563,156.705
C07939=1041.368,-75.434,424.285,169.032,35.563,156.705
C07940=1041.361,-75.684,424.296,169.030,35.563,156.705
C07941=1041.356,-75.934,424.307,169.028,35.563,156.705
C07942=1041.349,-76.183,424.319,169.025,35.562,156.705
C07943=1041.343,-76.433,424.330,169.023,35.562,156.705
C07944=1041.337,-76.683,424.341,169.020,35.562,156.705
C07945=1041.331,-76.933,424.352,169.018,35.562,156.705
C07946=1041.325,-77.182,424.364,169.016,35.561,156.705
C07947=1041.318,-77.432,424.375,169.013,35.561,156.705
C07948=1041.313,-77.682,424.386,169.011,35.561,156.705
C07949=1041.306,-77.931,424.398,169.009,35.561,156.705
C07950=1041.300,-78.181,424.409,169.006,35.560,156.705
C07951=1041.294,-78.431,424.420,169.004,35.560,156.705
C07952=1041.288,-78.680,424.431,169.002,35.560,156.705
C07953=1041.282,-78.931,424.442,168.999,35.560,156.705
C07954=1041.276,-79.180,424.454,168.997,35.559,156.705
C07955=1041.269,-79.430,424.465,168.994,35.559,156.705
C07956=1041.263,-79.679,424.475,168.992,35.559,156.705
C07957=1041.256,-79.929,424.486,168.990,35.559,156.705
C07958=1041.251,-80.179,424.497,168.987,35.559,156.705
C07959=1041.244,-80.429,424.509,168.985,35.559,156.705
C07960=1041.238,-80.677,424.520,168.982,35.559,156.705
C07961=1041.231,-80.928,424.531,168.980,35.558,156.705
C07962=1041.226,-81.177,424.542,168.978,35.558,156.705
C07963=1041.219,-81.427,424.553,168.975,35.558,156.705
C07964=1041.213,-81.676,424.563,168.973,35.558,156.705
C07965=1041.206,-81.927,424.574,168.970,35.558,156.705
C07966=1041.201,-82.176,424.585,168.968,35.558,156.705
C07967=1041.194,-82.425,424.596,168.966,35.558,156.705
C07968=1041.188,-82.675,424.607,168.963,35.558,156.705
C07969=1041.182,-82.925,424.618,168.961,35.558,156.705
C07970=1041.175,-83.175,424.628,168.958,35.558,156.705
C07971=1041.168,-83.459,424.641,168.956,35.558,156.705
C07972=1041.161,-83.744,424.654,168.953,35.557,156.705
C07973=1041.154,-84.030,424.666,168.950,35.557,156.705
C07974=1041.147,-84.314,424.678,168.947,35.557,156.705
C07975=1041.140,-84.564,424.689,168.945,35.557,156.705
C07976=1041.135,-84.814,424.700,168.942,35.557,156.705
C07977=1041.129,-85.063,424.711,168.940,35.557,156.705
C07978=1041.122,-85.313,424.721,168.938,35.557,156.705
C07979=1041.116,-85.563,424.732,168.935,35.557,156.705
C07980=1041.110,-85.813,424.743,168.933,35.557,156.705
C07981=1041.103,-86.062,424.754,168.930,35.557,156.705
C07982=1041.097,-86.312,424.765,168.928,35.557,156.705
C07983=1041.091,-86.562,424.776,168.925,35.557,156.706
C07984=1041.085,-86.811,424.786,168.923,35.557,156.706
C07985=1041.079,-87.060,424.797,168.921,35.557,156.706
C07986=1041.073,-87.311,424.808,168.918,35.557,156.706
C07987=1041.066,-87.560,424.818,168.916,35.557,156.706
C07988=1041.060,-87.810,424.830,168.913,35.556,156.706
C07989=1041.053,-88.059,424.840,168.911,35.556,156.706
C07990=1041.048,-88.309,424.850,168.908,35.556,156.706
C07991=1041.042,-88.559,424.861,168.906,35.556,156.706
C07992=1041.035,-88.809,424.872,168.904,35.556,156.706
C07993=1041.029,-89.058,424.883,168.901,35.556,156.706
C07994=1041.023,-89.308,424.893,168.899,35.556,156.706
C07995=1041.016,-89.557,424.904,168.896,35.556,156.706
C07996=1041.011,-89.808,424.914,168.894,35.556,156.706
C07997=1041.005,-90.057,424.925,168.891,35.556,156.706
C07998=1040.998,-90.307,424.936,168.889,35.556,156.706
C07999=1040.992,-90.556,424.947,168.886,35.556,156.706
C08000=1040.986,-90.806,424.957,168.884,35.556,156.706
C08001=1040.981,-91.056,424.967,168.882,35.556,156.706
C08002=1040.974,-91.306,424.978,168.879,35.556,156.706
C08003=1040.968,-91.555,424.989,168.877,35.556,156.706
C08004=1040.962,-91.805,424.999,168.874,35.556,156.706
C08005=1040.956,-92.054,425.009,168.872,35.556,156.706
C08006=1040.949,-92.305,425.020,168.869,35.556,156.706
C08007=1040.944,-92.554,425.031,168.868,35.556,156.706
C08008=1040.937,-92.803,425.041,168.865,35.556,156.706
C08009=1040.932,-93.053,425.052,168.863,35.556,156.706
C08010=1040.925,-93.303,425.062,168.861,35.556,156.706
C08011=1040.919,-93.553,425.073,168.858,35.556,156.706
C08012=1040.914,-93.803,425.083,168.856,35.556,156.706
C08013=1040.907,-94.052,425.094,168.853,35.556,156.706
C08014=1040.901,-94.302,425.104,168.851,35.556,156.706
C08015=1040.895,-94.552,425.114,168.848,35.556,156.706
C08016=1040.889,-94.802,425.125,168.846,35.556,156.706
C08017=1040.882,-95.051,425.136,168.843,35.556,156.706
C08018=1040.877,-95.301,425.146,168.841,35.556,156.706
C08019=1040.871,-95.550,425.157,168.839,35.556,156.706
C08020=1040.865,-95.799,425.167,168.836,35.556,156.706
C08021=1040.859,-96.050,425.177,168.834,35.556,156.706
C08022=1040.852,-96.299,425.188,168.831,35.556,156.706
C08023=1040.847,-96.550,425.198,168.829,35.556,156.706
C08024=1040.840,-96.799,425.208,168.826,35.556,156.706
C08025=1040.835,-97.048,425.219,168.824,35.556,156.706
C08026=1040.829,-97.298,425.229,168.821,35.556,156.706
C08027=1040.823,-97.548,425.239,168.819,35.557,156.707
C08028=1040.816,-97.798,425.249,168.816,35.557,156.707
C08029=1040.810,-98.048,425.260,168.814,35.557,156.707
C08030=1040.804,-98.297,425.270,168.811,35.556,156.707
C08031=1040.797,-98.546,425.280,168.809,35.557,156.707
C08032=1040.792,-98.797,425.290,168.806,35.557,156.707
C08033=1040.786,-99.046,425.301,168.804,35.557,156.707
C08034=1040.779,-99.296,425.310,168.801,35.558,156.707
C08035=1040.773,-99.583,425.322,168.799,35.557,156.707
C08036=1040.765,-99.870,425.334,168.796,35.558,156.707
C08037=1040.758,-100.157,425.345,168.793,35.558,156.707
C08038=1040.751,-100.445,425.357,168.790,35.558,156.707
C08039=1040.745,-100.694,425.367,168.787,35.558,156.707
C08040=1040.739,-100.944,425.377,168.785,35.558,156.707
C08041=1040.733,-101.194,425.387,168.782,35.558,156.707
C08042=1040.727,-101.443,425.397,168.780,35.559,156.707
C08043=1040.720,-101.694,425.407,168.777,35.559,156.707
C08044=1040.714,-101.943,425.418,168.775,35.559,156.708
C08045=1040.708,-102.193,425.428,168.772,35.559,156.708
C08046=1040.702,-102.443,425.437,168.770,35.559,156.708
C08047=1040.696,-102.692,425.448,168.767,35.560,156.708
C08048=1040.690,-102.942,425.458,168.765,35.560,156.708
C08049=1040.684,-103.192,425.467,168.762,35.560,156.708
C08050=1040.677,-103.441,425.477,168.760,35.560,156.708
C08051=1040.672,-103.691,425.488,168.757,35.560,156.708
C08052=1040.666,-103.941,425.497,168.756,35.561,156.708
C08053=1040.660,-104.191,425.507,168.753,35.561,156.708
C08054=1040.653,-104.440,425.517,168.751,35.561,156.708
C08055=1040.648,-104.690,425.527,168.748,35.561,156.708
C08056=1040.641,-104.940,425.537,168.746,35.561,156.708
C08057=1040.635,-105.189,425.547,168.743,35.562,156.708
C08058=1040.629,-105.439,425.557,168.741,35.562,156.708
C08059=1040.623,-105.689,425.567,168.738,35.562,156.708
C08060=1040.617,-105.939,425.576,168.736,35.562,156.708
C08061=1040.611,-106.188,425.587,168.733,35.563,156.709
C08062=1040.605,-106.438,425.596,168.731,35.563,156.709
C08063=1040.599,-106.688,425.606,168.728,35.563,156.709
C08064=1040.593,-106.938,425.616,168.726,35.563,156.709
C08065=1040.587,-107.187,425.626,168.723,35.564,156.709
C08066=1040.581,-107.437,425.635,168.721,35.564,156.709
C08067=1040.574,-107.686,425.645,168.718,35.565,156.709
C08068=1040.568,-107.936,425.655,168.716,35.564,156.709
C08069=1040.562,-108.186,425.665,168.713,35.565,156.709
C08070=1040.556,-108.436,425.675,168.711,35.565,156.709
C08071=1040.550,-108.686,425.684,168.708,35.566,156.709
C08072=1040.544,-108.936,425.694,168.706,35.566,156.709
C08073=1040.538,-109.185,425.703,168.703,35.566,156.709
C08074=1040.532,-109.435,425.713,168.701,35.567,156.710
C08075=1040.525,-109.684,425.723,168.698,35.567,156.710
C08076=1040.519,-109.934,425.733,168.695,35.567,156.710
C08077=1040.513,-110.184,425.742,168.693,35.567,156.710
C08078=1040.507,-110.434,425.752,168.690,35.568,156.710
C08079=1040.501,-110.684,425.761,168.688,35.568,156.710
C08080=1040.495,-110.933,425.771,168.685,35.568,156.710
C08081=1040.489,-111.182,425.780,168.684,35.569,156.710
C08082=1040.483,-111.432,425.790,168.681,35.569,156.710
C08083=1040.476,-111.682,425.799,168.679,35.569,156.710
C08084=1040.471,-111.932,425.810,168.676,35.570,156.710
C08085=1040.465,-112.182,425.819,168.674,35.570,156.710
C08086=1040.459,-112.432,425.829,168.671,35.570,156.711
C08087=1040.452,-112.682,425.838,168.668,35.571,156.711
C08088=1040.446,-112.931,425.848,168.666,35.571,156.711
C08089=1040.441,-113.180,425.857,168.663,35.572,156.711
C08090=1040.435,-113.430,425.867,168.661,35.572,156.711
C08091=1040.428,-113.680,425.876,168.658,35.572,156.711
C08092=1040.422,-113.930,425.886,168.656,35.573,156.711
C08093=1040.416,-114.180,425.895,168.653,35.573,156.711
C08094=1040.410,-114.430,425.904,168.651,35.573,156.711
C08095=1040.404,-114.680,425.914,168.648,35.574,156.711
C08096=1040.398,-114.929,425.923,168.646,35.574,156.711
C08097=1040.392,-115.179,425.932,168.643,35.575,156.712
C08098=1040.386,-115.429,425.942,168.640,35.575,156.712
C08099=1040.379,-115.715,425.952,168.637,35.576,156.712
C08100=1040.372,-116.001,425.963,168.635,35.576,156.712
C08101=1040.365,-116.287,425.975,168.632,35.577,156.712
C08102=1040.357,-116.574,425.985,168.629,35.577,156.712
C08103=1040.352,-116.823,425.994,168.627,35.578,156.712
C08104=1040.346,-117.073,426.003,168.625,35.578,156.712
C08105=1040.340,-117.323,426.013,168.622,35.578,156.712
C08106=1040.334,-117.573,426.022,168.619,35.579,156.712
C08107=1040.328,-117.823,426.032,168.617,35.580,156.713
C08108=1040.322,-118.072,426.041,168.614,35.580,156.713
C08109=1040.315,-118.322,426.049,168.612,35.580,156.713
C08110=1040.309,-118.572,426.059,168.609,35.581,156.713
C08111=1040.303,-118.821,426.068,168.607,35.581,156.713
C08112=1040.297,-119.071,426.078,168.604,35.582,156.713
C08113=1040.292,-119.321,426.086,168.601,35.582,156.713
C08114=1040.285,-119.571,426.096,168.599,35.583,156.713
C08115=1040.279,-119.821,426.106,168.596,35.583,156.713
C08116=1040.273,-120.070,426.113,168.594,35.584,156.714
C08117=1040.267,-120.320,426.123,168.591,35.584,156.714
C08118=1040.261,-120.570,426.133,168.589,35.585,156.714
C08119=1040.255,-120.819,426.142,168.586,35.585,156.714
C08120=1040.249,-121.069,426.151,168.583,35.586,156.714
C08121=1040.243,-121.319,426.160,168.581,35.587,156.714
C08122=1040.236,-121.568,426.169,168.579,35.587,156.714
C08123=1040.230,-121.819,426.178,168.577,35.587,156.714
C08124=1040.225,-122.068,426.187,168.574,35.588,156.714
C08125=1040.219,-122.318,426.196,168.571,35.588,156.715
C08126=1040.213,-122.568,426.206,168.569,35.589,156.715
C08127=1040.207,-122.817,426.215,168.566,35.589,156.715
C08128=1040.201,-123.067,426.223,168.564,35.590,156.715
C08129=1040.195,-123.317,426.233,168.561,35.591,156.715
C08130=1040.189,-123.567,426.241,168.559,35.591,156.715
C08131=1040.183,-123.817,426.251,168.556,35.592,156.715
C08132=1040.176,-124.066,426.260,168.553,35.592,156.715
C08133=1040.170,-124.316,426.269,168.551,35.593,156.716
C08134=1040.165,-124.566,426.278,168.548,35.594,156.716
C08135=1040.159,-124.816,426.287,168.546,35.594,156.716
C08136=1040.152,-125.065,426.296,168.543,35.595,156.716
C08137=1040.147,-125.315,426.304,168.540,35.595,156.716
C08138=1040.141,-125.565,426.314,168.538,35.596,156.716
C08139=1040.134,-125.815,426.322,168.535,35.597,156.716
C08140=1040.128,-126.064,426.331,168.534,35.597,156.716
C08141=1040.123,-126.315,426.340,168.531,35.598,156.717
C08142=1040.116,-126.563,426.349,168.528,35.598,156.717
C08143=1040.110,-126.814,426.357,168.526,35.599,156.717
C08144=1040.104,-127.064,426.367,168.523,35.599,156.717
C08145=1040.098,-127.313,426.375,168.521,35.600,156.717
C08146=1040.092,-127.563,426.384,168.518,35.601,156.717
C08147=1040.087,-127.813,426.393,168.515,35.601,156.717
C08148=1040.081,-128.062,426.402,168.513,35.602,156.717
C08149=1040.076,-128.312,426.412,168.511,35.602,156.717
C08150=1040.073,-128.562,426.423,168.508,35.601,156.717
C08151=1040.070,-128.812,426.433,168.506,35.600,156.717
C08152=1040.067,-129.061,426.445,168.504,35.598,156.717
C08153=1040.066,-129.312,426.458,168.503,35.596,156.717
C08154=1040.066,-129.561,426.471,168.500,35.594,156.716
C08155=1040.066,-129.812,426.484,168.498,35.591,156.716
C08156=1040.067,-130.061,426.498,168.497,35.587,156.715
C08157=1040.068,-130.312,426.513,168.496,35.584,156.715
C08158=1040.072,-130.562,426.528,168.494,35.579,156.714
C08159=1040.076,-130.812,426.544,168.493,35.575,156.713
C08160=1040.080,-131.063,426.561,168.492,35.569,156.712
C08161=1040.085,-131.313,426.577,168.491,35.563,156.711
C08162=1040.090,-131.562,426.595,168.490,35.558,156.710
C08163=1039.746,-131.587,426.335,168.442,35.755,156.744
C08164=1039.739,-131.337,426.317,168.444,35.761,156.745
C08165=1039.734,-131.087,426.300,168.444,35.766,156.746
C08166=1039.730,-130.837,426.284,168.446,35.772,156.747
C08167=1039.726,-130.586,426.268,168.447,35.777,156.748
C08168=1039.724,-130.336,426.252,168.448,35.781,156.748
C08169=1039.722,-130.087,426.237,168.450,35.785,156.749
C08170=1039.720,-129.835,426.223,168.452,35.788,156.749
C08171=1039.721,-129.585,426.210,168.453,35.791,156.750
C08172=1039.721,-129.336,426.196,168.455,35.793,156.750
C08173=1039.722,-129.086,426.184,168.456,35.795,156.751
C08174=1039.724,-128.836,426.173,168.459,35.797,156.751
C08175=1039.727,-128.586,426.162,168.461,35.798,156.751
C08176=1039.731,-128.336,426.151,168.464,35.799,156.751
C08177=1039.735,-128.086,426.141,168.466,35.799,156.751
C08178=1039.740,-127.837,426.131,168.468,35.799,156.751
C08179=1039.746,-127.588,426.123,168.471,35.798,156.751
C08180=1039.752,-127.338,426.114,168.473,35.798,156.751
C08181=1039.758,-127.087,426.105,168.475,35.797,156.751
C08182=1039.765,-126.839,426.096,168.478,35.796,156.751
C08183=1039.771,-126.588,426.087,168.480,35.795,156.750
C08184=1039.776,-126.338,426.079,168.483,35.795,156.750
C08185=1039.783,-126.089,426.070,168.486,35.794,156.750
C08186=1039.789,-125.839,426.061,168.488,35.793,156.750
C08187=1039.794,-125.589,426.052,168.491,35.793,156.750
C08188=1039.801,-125.339,426.044,168.494,35.792,156.750
C08189=1039.807,-125.090,426.034,168.496,35.792,156.750
C08190=1039.812,-124.840,426.026,168.499,35.791,156.750
C08191=1039.819,-124.590,426.017,168.501,35.790,156.749
C08192=1039.825,-124.340,426.008,168.504,35.790,156.749
C08193=1039.831,-124.091,425.999,168.507,35.789,156.749
C08194=1039.837,-123.841,425.989,168.509,35.789,156.749
C08195=1039.843,-123.591,425.981,168.512,35.788,156.749
C08196=1039.849,-123.342,425.972,168.513,35.787,156.749
C08197=1039.855,-123.091,425.963,168.516,35.787,156.749
C08198=1039.861,-122.842,425.953,168.519,35.786,156.749
C08199=1039.866,-122.592,425.945,168.521,35.785,156.748
C08200=1039.873,-122.342,425.936,168.524,35.785,156.748
C08201=1039.879,-122.093,425.926,168.526,35.784,156.748
C08202=1039.885,-121.842,425.917,168.529,35.784,156.748
C08203=1039.891,-121.593,425.908,168.532,35.783,156.748
C08204=1039.897,-121.343,425.899,168.534,35.782,156.748
C08205=1039.903,-121.093,425.890,168.537,35.782,156.748
C08206=1039.909,-120.844,425.881,168.539,35.781,156.748
C08207=1039.915,-120.594,425.871,168.542,35.781,156.748
C08208=1039.921,-120.344,425.863,168.545,35.781,156.747
C08209=1039.927,-120.094,425.853,168.547,35.780,156.747
C08210=1039.933,-119.845,425.844,168.550,35.780,156.747
C08211=1039.939,-119.595,425.836,168.552,35.779,156.747
C08212=1039.946,-119.345,425.826,168.555,35.778,156.747
C08213=1039.952,-119.095,425.816,168.558,35.778,156.747
C08214=1039.957,-118.846,425.807,168.559,35.777,156.747
C08215=1039.963,-118.596,425.798,168.562,35.776,156.747
C08216=1039.969,-118.346,425.789,168.564,35.777,156.747
C08217=1039.976,-118.096,425.779,168.567,35.776,156.746
C08218=1039.982,-117.847,425.770,168.570,35.775,156.746
C08219=1039.988,-117.597,425.762,168.572,35.775,156.746
C08220=1039.994,-117.347,425.752,168.575,35.774,156.746
C08221=1040.000,-117.097,425.743,168.577,35.774,156.746
C08222=1040.006,-116.848,425.733,168.580,35.774,156.746
C08223=1040.012,-116.598,425.724,168.582,35.773,156.746
C08224=1040.019,-116.312,425.713,168.585,35.772,156.746
C08225=1040.026,-116.026,425.703,168.588,35.772,156.746
C08226=1040.033,-115.739,425.692,168.591,35.771,156.745
C08227=1040.039,-115.452,425.681,168.594,35.771,156.745
C08228=1040.046,-115.203,425.672,168.597,35.770,156.745
C08229=1040.052,-114.953,425.663,168.599,35.770,156.745
C08230=1040.058,-114.704,425.653,168.602,35.769,156.745
C08231=1040.064,-114.454,425.644,168.605,35.769,156.745
C08232=1040.070,-114.204,425.634,168.607,35.768,156.745
C08233=1040.077,-113.955,425.625,168.609,35.768,156.745
C08234=1040.082,-113.704,425.616,168.611,35.768,156.745
C08235=1040.089,-113.454,425.606,168.614,35.767,156.745
C08236=1040.095,-113.205,425.597,168.616,35.766,156.744
C08237=1040.100,-112.956,425.587,168.619,35.767,156.744
C08238=1040.107,-112.706,425.578,168.621,35.766,156.744
C08239=1040.112,-112.456,425.568,168.624,35.765,156.744
C08240=1040.118,-112.206,425.558,168.627,35.765,156.744
C08241=1040.124,-111.956,425.549,168.629,35.765,156.744
C08242=1040.130,-111.706,425.539,168.632,35.764,156.744
C08243=1040.137,-111.456,425.529,168.634,35.764,156.744
C08244=1040.143,-111.207,425.520,168.637,35.764,156.744
C08245=1040.149,-110.957,425.510,168.639,35.763,156.744
C08246=1040.155,-110.708,425.501,168.642,35.763,156.744
C08247=1040.161,-110.458,425.492,168.645,35.762,156.744
C08248=1040.167,-110.208,425.482,168.647,35.762,156.743
C08249=1040.173,-109.958,425.472,168.650,35.762,156.743
C08250=1040.179,-109.709,425.463,168.652,35.761,156.743
C08251=1040.186,-109.459,425.453,168.655,35.761,156.743
C08252=1040.192,-109.210,425.443,168.657,35.761,156.743
C08253=1040.198,-108.960,425.433,168.660,35.760,156.743
C08254=1040.203,-108.710,425.423,168.662,35.760,156.743
C08255=1040.210,-108.460,425.414,168.665,35.760,156.743
C08256=1040.216,-108.210,425.404,168.666,35.759,156.743
C08257=1040.222,-107.960,425.395,168.669,35.759,156.743
C08258=1040.228,-107.710,425.385,168.672,35.758,156.743
C08259=1040.234,-107.461,425.375,168.674,35.758,156.742
C08260=1040.241,-107.212,425.365,168.677,35.758,156.742
C08261=1040.247,-106.962,425.356,168.679,35.757,156.742
C08262=1040.252,-106.712,425.345,168.682,35.757,156.742
C08263=1040.259,-106.462,425.336,168.684,35.757,156.742
C08264=1040.265,-106.212,425.326,168.687,35.757,156.742
C08265=1040.271,-105.963,425.316,168.689,35.756,156.742
C08266=1040.277,-105.713,425.306,168.692,35.756,156.742
C08267=1040.283,-105.463,425.296,168.694,35.756,156.742
C08268=1040.289,-105.213,425.287,168.697,35.756,156.742
C08269=1040.296,-104.964,425.276,168.699,35.755,156.742
C08270=1040.302,-104.714,425.267,168.702,35.755,156.742
C08271=1040.307,-104.464,425.257,168.704,35.755,156.742
C08272=1040.313,-104.214,425.247,168.707,35.755,156.742
C08273=1040.320,-103.965,425.237,168.710,35.755,156.742
C08274=1040.326,-103.715,425.227,168.712,35.754,156.742
C08275=1040.331,-103.465,425.217,168.715,35.754,156.742
C08276=1040.338,-103.216,425.207,168.717,35.753,156.741
C08277=1040.344,-102.966,425.197,168.720,35.754,156.741
C08278=1040.349,-102.716,425.187,168.722,35.753,156.741
C08279=1040.356,-102.467,425.177,168.725,35.753,156.741
C08280=1040.362,-102.217,425.167,168.727,35.752,156.741
C08281=1040.368,-101.967,425.158,168.730,35.752,156.741
C08282=1040.374,-101.718,425.147,168.732,35.752,156.741
C08283=1040.380,-101.468,425.137,168.735,35.752,156.741
C08284=1040.386,-101.218,425.128,168.737,35.752,156.741
C08285=1040.393,-100.968,425.116,168.740,35.751,156.741
C08286=1040.399,-100.718,425.107,168.742,35.751,156.741
C08287=1040.405,-100.469,425.097,168.745,35.751,156.741
C08288=1040.412,-100.181,425.085,168.747,35.751,156.741
C08289=1040.419,-99.894,425.074,168.750,35.751,156.741
C08290=1040.426,-99.607,425.063,168.752,35.750,156.741
C08291=1040.433,-99.320,425.050,168.755,35.750,156.741
C08292=1040.439,-99.071,425.041,168.758,35.750,156.740
C08293=1040.446,-98.821,425.030,168.760,35.750,156.740
C08294=1040.451,-98.571,425.020,168.763,35.750,156.740
C08295=1040.458,-98.321,425.009,168.765,35.749,156.740
C08296=1040.464,-98.072,425.000,168.768,35.749,156.740
C08297=1040.470,-97.822,424.989,168.770,35.749,156.740
C08298=1040.476,-97.572,424.979,168.773,35.749,156.740
C08299=1040.482,-97.322,424.968,168.775,35.749,156.740
C08300=1040.489,-97.072,424.959,168.778,35.749,156.740
C08301=1040.494,-96.823,424.948,168.780,35.749,156.740
C08302=1040.500,-96.573,424.938,168.783,35.748,156.740
C08303=1040.506,-96.324,424.927,168.785,35.748,156.740
C08304=1040.512,-96.074,424.918,168.788,35.748,156.740
C08305=1040.518,-95.824,424.907,168.790,35.748,156.740
C08306=1040.525,-95.575,424.897,168.793,35.748,156.740
C08307=1040.531,-95.324,424.886,168.795,35.749,156.740
C08308=1040.536,-95.075,424.875,168.798,35.748,156.740
C08309=1040.543,-94.826,424.865,168.800,35.748,156.740
C08310=1040.548,-94.576,424.855,168.802,35.748,156.740
C08311=1040.555,-94.326,424.844,168.805,35.748,156.740
C08312=1040.561,-94.076,424.833,168.807,35.748,156.740
C08313=1040.567,-93.826,424.824,168.810,35.748,156.740
C08314=1040.573,-93.577,424.813,168.812,35.748,156.740
C08315=1040.579,-93.327,424.802,168.815,35.748,156.740
C08316=1040.585,-93.078,424.792,168.817,35.748,156.740
C08317=1040.591,-92.827,424.781,168.820,35.748,156.740
C08318=1040.598,-92.578,424.771,168.822,35.748,156.740
C08319=1040.603,-92.328,424.761,168.825,35.748,156.740
C08320=1040.609,-92.079,424.750,168.827,35.748,156.740
C08321=1040.615,-91.829,424.739,168.830,35.747,156.739
C08322=1040.622,-91.579,424.728,168.832,35.747,156.739
C08323=1040.628,-91.330,424.719,168.834,35.747,156.739
C08324=1040.634,-91.080,424.708,168.837,35.747,156.739
C08325=1040.640,-90.830,424.697,168.839,35.747,156.739
C08326=1040.646,-90.581,424.686,168.842,35.748,156.739
C08327=1040.652,-90.331,424.676,168.844,35.748,156.739
C08328=1040.658,-90.081,424.665,168.847,35.748,156.739
C08329=1040.665,-89.831,424.655,168.849,35.748,156.739
C08330=1040.670,-89.582,424.644,168.852,35.748,156.739
C08331=1040.677,-89.333,424.633,168.854,35.747,156.739
C08332=1040.683,-89.082,424.622,168.857,35.747,156.739
C08333=1040.689,-88.832,424.612,168.859,35.747,156.739
C08334=1040.695,-88.583,424.602,168.861,35.747,156.739
C08335=1040.701,-88.334,424.591,168.864,35.747,156.739
C08336=1040.707,-88.083,424.580,168.866,35.747,156.739
C08337=1040.714,-87.834,424.569,168.869,35.747,156.739
C08338=1040.719,-87.585,424.558,168.871,35.747,156.739
C08339=1040.727,-87.335,424.548,168.874,35.748,156.739
C08340=1040.732,-87.085,424.538,168.876,35.748,156.739
C08341=1040.738,-86.835,424.527,168.879,35.748,156.739
C08342=1040.745,-86.585,424.516,168.881,35.748,156.739
C08343=1040.751,-86.336,424.505,168.883,35.748,156.739
C08344=1040.757,-86.086,424.494,168.886,35.747,156.739
C08345=1040.763,-85.836,424.484,168.887,35.747,156.739
C08346=1040.769,-85.587,424.473,168.890,35.747,156.739
C08347=1040.775,-85.337,424.462,168.892,35.747,156.739
C08348=1040.782,-85.088,424.451,168.895,35.747,156.739
C08349=1040.788,-84.837,424.440,168.897,35.747,156.739
C08350=1040.794,-84.588,424.429,168.900,35.747,156.739
C08351=1040.800,-84.339,424.419,168.902,35.747,156.739
C08352=1040.808,-84.053,424.407,168.905,35.748,156.739
C08353=1040.815,-83.768,424.394,168.907,35.748,156.739
C08354=1040.821,-83.484,424.381,168.910,35.748,156.739
C08355=1040.829,-83.198,424.369,168.913,35.748,156.739
C08356=1040.835,-82.949,424.358,168.915,35.748,156.739
C08357=1040.842,-82.699,424.347,168.918,35.748,156.739
C08358=1040.847,-82.449,424.336,168.920,35.748,156.739
C08359=1040.854,-82.200,424.326,168.923,35.748,156.739
C08360=1040.860,-81.950,424.315,168.925,35.748,156.739
C08361=1040.866,-81.700,424.304,168.928,35.748,156.739
C08362=1040.873,-81.451,424.293,168.930,35.748,156.739
C08363=1040.879,-81.201,424.282,168.932,35.748,156.739
C08364=1040.885,-80.951,424.271,168.935,35.748,156.739
C08365=1040.891,-80.702,424.260,168.937,35.748,156.739
C08366=1040.898,-80.452,424.249,168.940,35.748,156.739
C08367=1040.904,-80.203,424.238,168.942,35.748,156.739
C08368=1040.910,-79.953,424.227,168.945,35.748,156.739
C08369=1040.917,-79.703,424.216,168.947,35.748,156.739
C08370=1040.923,-79.453,424.205,168.949,35.748,156.739
C08371=1040.929,-79.204,424.194,168.952,35.749,156.739
C08372=1040.935,-78.954,424.182,168.954,35.749,156.739
C08373=1040.941,-78.705,424.172,168.957,35.749,156.739
C08374=1040.948,-78.455,424.160,168.959,35.749,156.739
C08375=1040.953,-78.205,424.149,168.961,35.749,156.739
C08376=1040.960,-77.955,424.137,168.964,35.750,156.739
C08377=1040.966,-77.706,424.127,168.966,35.750,156.739
C08378=1040.972,-77.456,424.115,168.968,35.750,156.739
C08379=1040.978,-77.206,424.104,168.971,35.750,156.739
C08380=1040.984,-76.957,424.093,168.973,35.750,156.739
C08381=1040.990,-76.707,424.082,168.976,35.751,156.739
C08382=1040.996,-76.457,424.070,168.978,35.751,156.739
C08383=1041.003,-76.207,424.058,168.980,35.751,156.739
C08384=1041.009,-75.958,424.048,168.983,35.751,156.739
C08385=1041.015,-75.708,424.036,168.985,35.751,156.739
C08386=1041.021,-75.458,424.025,168.988,35.752,156.739
C08387=1041.028,-75.209,424.014,168.990,35.752,156.739
C08388=1041.034,-74.960,424.003,168.992,35.752,156.739
C08389=1041.041,-74.710,423.991,168.995,35.752,156.739
C08390=1041.046,-74.460,423.980,168.997,35.753,156.739
C08391=1041.053,-74.210,423.969,168.999,35.753,156.739
C08392=1041.059,-73.961,423.957,169.002,35.753,156.739
C08393=1041.064,-73.711,423.946,169.004,35.753,156.739
C08394=1041.071,-73.461,423.934,169.006,35.753,156.739
C08395=1041.077,-73.212,423.923,169.009,35.753,156.739
C08396=1041.083,-72.962,423.912,169.011,35.754,156.739
C08397=1041.089,-72.713,423.900,169.013,35.754,156.739
C08398=1041.095,-72.462,423.888,169.017,35.755,156.739
C08399=1041.101,-72.213,423.877,169.019,35.755,156.739
C08400=1041.107,-71.963,423.865,169.021,35.755,156.739
C08401=1041.114,-71.714,423.853,169.024,35.756,156.739
C08402=1041.119,-71.464,423.842,169.026,35.756,156.739
C08403=1041.125,-71.214,423.830,169.028,35.756,156.739
C08404=1041.131,-70.965,423.819,169.031,35.756,156.739
C08405=1041.138,-70.715,423.807,169.033,35.757,156.739
C08406=1041.143,-70.465,423.795,169.035,35.757,156.739
C08407=1041.149,-70.216,423.784,169.038,35.758,156.740
C08408=1041.156,-69.966,423.772,169.040,35.758,156.740
C08409=1041.162,-69.717,423.761,169.042,35.758,156.739
C08410=1041.169,-69.467,423.749,169.045,35.759,156.740
C08411=1041.174,-69.217,423.737,169.047,35.759,156.740
C08412=1041.180,-68.968,423.725,169.049,35.759,156.740
C08413=1041.187,-68.718,423.714,169.052,35.759,156.740
C08414=1041.193,-68.468,423.702,169.054,35.760,156.740
C08415=1041.198,-68.219,423.690,169.056,35.760,156.740
C08416=1041.206,-67.936,423.677,169.059,35.761,156.740
C08417=1041.213,-67.653,423.664,169.062,35.761,156.740
C08418=1041.219,-67.370,423.651,169.064,35.762,156.740
C08419=1041.226,-67.088,423.637,169.067,35.762,156.740
C08420=1041.233,-66.838,423.626,169.069,35.762,156.740
C08421=1041.239,-66.588,423.614,169.071,35.762,156.740
C08422=1041.245,-66.339,423.602,169.074,35.763,156.740
C08423=1041.251,-66.089,423.590,169.076,35.763,156.740
C08424=1041.258,-65.839,423.578,169.078,35.764,156.740
C08425=1041.263,-65.590,423.566,169.081,35.764,156.740
C08426=1041.269,-65.340,423.555,169.083,35.765,156.740
C08427=1041.276,-65.090,423.543,169.085,35.765,156.740
C08428=1041.283,-64.841,423.531,169.088,35.765,156.740
C08429=1041.288,-64.592,423.519,169.090,35.765,156.740
C08430=1041.294,-64.342,423.508,169.092,35.766,156.741
C08431=1041.301,-64.092,423.496,169.094,35.766,156.740
C08432=1041.307,-63.842,423.483,169.097,35.767,156.741
C08433=1041.313,-63.593,423.471,169.099,35.767,156.741
C08434=1041.319,-63.343,423.460,169.101,35.768,156.741
C08435=1041.326,-63.093,423.448,169.104,35.768,156.741
C08436=1041.332,-62.844,423.436,169.106,35.768,156.741
C08437=1041.338,-62.595,423.424,169.108,35.768,156.741
C08438=1041.344,-62.345,423.412,169.111,35.769,156.741
C08439=1041.350,-62.095,423.400,169.113,35.769,156.741
C08440=1041.357,-61.845,423.388,169.115,35.770,156.741
C08441=1041.363,-61.595,423.376,169.117,35.770,156.741
C08442=1041.369,-61.346,423.364,169.120,35.770,156.741
C08443=1041.375,-61.097,423.352,169.122,35.770,156.741
C08444=1041.382,-60.847,423.340,169.124,35.771,156.741
C08445=1041.388,-60.597,423.328,169.127,35.772,156.741
C08446=1041.394,-60.347,423.317,169.129,35.772,156.741
C08447=1041.401,-60.097,423.305,169.131,35.773,156.741
C08448=1041.406,-59.848,423.292,169.133,35.773,156.741
C08449=1041.413,-59.599,423.280,169.137,35.773,156.741
C08450=1041.419,-59.349,423.268,169.139,35.773,156.741
C08451=1041.425,-59.099,423.256,169.141,35.774,156.742
C08452=1041.432,-58.850,423.244,169.144,35.774,156.742
C08453=1041.439,-58.600,423.232,169.146,35.775,156.742
C08454=1041.445,-58.350,423.219,169.148,35.775,156.742
C08455=1041.451,-58.101,423.208,169.150,35.776,156.742
C08456=1041.457,-57.851,423.197,169.153,35.776,156.742
C08457=1041.463,-57.601,423.184,169.155,35.776,156.742
C08458=1041.469,-57.352,423.172,169.157,35.777,156.742
C08459=1041.476,-57.102,423.160,169.160,35.777,156.742
C08460=1041.482,-56.852,423.148,169.162,35.778,156.742
C08461=1041.489,-56.603,423.136,169.164,35.778,156.742
C08462=1041.495,-56.353,423.124,169.166,35.778,156.742
C08463=1041.501,-56.103,423.111,169.169,35.779,156.742
C08464=1041.508,-55.854,423.099,169.171,35.779,156.742
C08465=1041.514,-55.605,423.088,169.173,35.780,156.742
C08466=1041.520,-55.355,423.075,169.176,35.780,156.742
C08467=1041.527,-55.106,423.062,169.178,35.781,156.742
C08468=1041.533,-54.856,423.050,169.180,35.781,156.742
C08469=1041.539,-54.607,423.038,169.182,35.781,156.742
C08470=1041.546,-54.357,423.026,169.185,35.782,156.743
C08471=1041.552,-54.107,423.013,169.187,35.782,156.743
C08472=1041.559,-53.857,423.001,169.189,35.783,156.743
C08473=1041.565,-53.608,422.989,169.191,35.783,156.743
C08474=1041.571,-53.358,422.977,169.194,35.783,156.743
C08475=1041.578,-53.108,422.965,169.196,35.784,156.743
C08476=1041.584,-52.859,422.952,169.198,35.784,156.743
C08477=1041.590,-52.609,422.940,169.200,35.785,156.743
C08478=1041.597,-52.360,422.928,169.203,35.785,156.743
C08479=1041.603,-52.110,422.915,169.205,35.786,156.743
C08480=1041.610,-51.828,422.901,169.207,35.786,156.743
C08481=1041.618,-51.547,422.888,169.210,35.786,156.743
C08482=1041.625,-51.266,422.874,169.213,35.787,156.743
C08483=1041.632,-50.984,422.860,169.215,35.788,156.743
C08484=1041.639,-50.735,422.848,169.217,35.788,156.743
C08485=1041.645,-50.485,422.835,169.220,35.788,156.743
C08486=1041.651,-50.236,422.822,169.222,35.789,156.744
C08487=1041.657,-49.986,422.810,169.225,35.790,156.744
C08488=1041.663,-49.736,422.798,169.227,35.790,156.744
C08489=1041.669,-49.486,422.785,169.229,35.791,156.744
C08490=1041.676,-49.237,422.772,169.232,35.791,156.744
C08491=1041.682,-48.987,422.760,169.234,35.792,156.744
C08492=1041.688,-48.737,422.747,169.236,35.793,156.744
C08493=1041.694,-48.488,422.734,169.238,35.793,156.744
C08494=1041.701,-48.239,422.722,169.240,35.794,156.744
C08495=1041.707,-47.989,422.709,169.243,35.794,156.744
C08496=1041.713,-47.739,422.696,169.245,35.795,156.744
C08497=1041.719,-47.490,422.684,169.247,35.795,156.744
C08498=1041.726,-47.240,422.672,169.249,35.796,156.745
C08499=1041.732,-46.991,422.658,169.251,35.797,156.745
C08500=1041.738,-46.741,422.646,169.254,35.797,156.745
C08501=1041.744,-46.492,422.633,169.256,35.798,156.745
C08502=1041.751,-46.242,422.621,169.258,35.799,156.745
C08503=1041.757,-45.991,422.608,169.260,35.799,156.745
C08504=1041.763,-45.742,422.594,169.262,35.799,156.745
C08505=1041.769,-45.492,422.582,169.265,35.800,156.745
C08506=1041.776,-45.243,422.569,169.267,35.801,156.745
C08507=1041.782,-44.993,422.557,169.269,35.802,156.745
C08508=1041.788,-44.744,422.543,169.271,35.802,156.745
C08509=1041.794,-44.494,422.531,169.273,35.803,156.746
C08510=1041.800,-44.245,422.517,169.275,35.804,156.746
C08511=1041.807,-43.996,422.506,169.278,35.804,156.746
C08512=1041.813,-43.746,422.493,169.281,35.804,156.746
C08513=1041.819,-43.496,422.480,169.283,35.805,156.746
C08514=1041.826,-43.246,422.467,169.285,35.806,156.746
C08515=1041.833,-42.997,422.454,169.287,35.806,156.746
C08516=1041.839,-42.747,422.442,169.290,35.807,156.746
C08517=1041.845,-42.498,422.428,169.292,35.808,156.746
C08518=1041.851,-42.248,422.415,169.294,35.808,156.746
C08519=1041.857,-41.999,422.402,169.296,35.809,156.747
C08520=1041.864,-41.750,422.390,169.298,35.809,156.746
C08521=1041.870,-41.499,422.377,169.300,35.810,156.747
C08522=1041.877,-41.250,422.364,169.303,35.810,156.747
C08523=1041.882,-41.000,422.351,169.305,35.811,156.747
C08524=1041.889,-40.751,422.338,169.307,35.812,156.747
C08525=1041.895,-40.501,422.326,169.309,35.813,156.747
C08526=1041.902,-40.252,422.313,169.311,35.813,156.747
C08527=1041.908,-40.002,422.299,169.313,35.814,156.747
C08528=1041.914,-39.752,422.286,169.316,35.815,156.747
C08529=1041.921,-39.503,422.273,169.318,35.815,156.747
C08530=1041.927,-39.253,422.260,169.320,35.815,156.747
C08531=1041.933,-39.004,422.248,169.322,35.816,156.748
C08532=1041.940,-38.754,422.234,169.324,35.817,156.748
C08533=1041.946,-38.504,422.222,169.326,35.817,156.748
C08534=1041.952,-38.255,422.208,169.328,35.818,156.748
C08535=1041.959,-38.005,422.195,169.332,35.819,156.748
C08536=1041.965,-37.756,422.182,169.334,35.819,156.748
C08537=1041.971,-37.506,422.169,169.336,35.821,156.748
C08538=1041.977,-37.256,422.156,169.338,35.821,156.748
C08539=1041.984,-37.007,422.142,169.340,35.822,156.748
C08540=1041.989,-36.757,422.129,169.342,35.823,156.749
C08541=1041.995,-36.508,422.116,169.344,35.823,156.749
C08542=1042.002,-36.258,422.102,169.346,35.824,156.749
C08543=1042.008,-36.008,422.089,169.349,35.825,156.749
C08544=1042.015,-35.728,422.075,169.351,35.825,156.749
C08545=1042.023,-35.447,422.060,169.353,35.826,156.749
C08546=1042.029,-35.165,422.045,169.356,35.827,156.749
C08547=1042.036,-34.885,422.030,169.358,35.828,156.749
C08548=1042.043,-34.635,422.016,169.360,35.829,156.750
C08549=1042.049,-34.386,422.003,169.362,35.829,156.750
C08550=1042.055,-34.136,421.991,169.364,35.830,156.750
C08551=1042.062,-33.886,421.977,169.367,35.831,156.750
C08552=1042.067,-33.636,421.963,169.369,35.832,156.750
C08553=1042.074,-33.387,421.950,169.372,35.832,156.750
C08554=1042.080,-33.138,421.937,169.374,35.833,156.750
C08555=1042.087,-32.888,421.923,169.376,35.834,156.750
C08556=1042.093,-32.639,421.910,169.378,35.835,156.750
C08557=1042.099,-32.389,421.897,169.380,35.836,156.751
C08558=1042.105,-32.139,421.884,169.382,35.836,156.751
C08559=1042.112,-31.889,421.870,169.384,35.837,156.751
C08560=1042.118,-31.640,421.857,169.387,35.838,156.751
C08561=1042.124,-31.391,421.844,169.389,35.838,156.751
C08562=1042.131,-31.141,421.830,169.391,35.839,156.751
C08563=1042.137,-30.892,421.817,169.393,35.840,156.751
C08564=1042.143,-30.642,421.803,169.395,35.840,156.751
C08565=1042.150,-30.392,421.789,169.397,35.841,156.751
C08566=1042.156,-30.143,421.776,169.399,35.842,156.752
C08567=1042.162,-29.894,421.763,169.401,35.843,156.752
C08568=1042.169,-29.644,421.749,169.403,35.844,156.752
C08569=1042.175,-29.394,421.736,169.405,35.844,156.752
C08570=1042.182,-29.144,421.722,169.408,35.845,156.752
C08571=1042.188,-28.895,421.709,169.411,35.846,156.752
C08572=1042.194,-28.646,421.696,169.413,35.846,156.752
C08573=1042.200,-28.396,421.681,169.415,35.847,156.752
C08574=1042.207,-28.146,421.668,169.417,35.848,156.753
C08575=1042.213,-27.897,421.655,169.419,35.848,156.753
C08576=1042.220,-27.647,421.641,169.421,35.849,156.753
C08577=1042.226,-27.398,421.628,169.423,35.850,156.753
C08578=1042.233,-27.148,421.614,169.425,35.851,156.753
C08579=1042.239,-26.899,421.601,169.427,35.852,156.753
C08580=1042.244,-26.649,421.587,169.429,35.852,156.753
C08581=1042.251,-26.399,421.574,169.431,35.853,156.753
C08582=1042.257,-26.150,421.560,169.433,35.854,156.754
C08583=1042.263,-25.901,421.546,169.436,35.855,156.754
C08584=1042.270,-25.651,421.532,169.438,35.856,156.754
C08585=1042.276,-25.402,421.519,169.440,35.856,156.754
C08586=1042.282,-25.151,421.505,169.442,35.858,156.754
C08587=1042.288,-24.902,421.491,169.445,35.858,156.754
C08588=1042.294,-24.653,421.477,169.447,35.859,156.754
C08589=1042.301,-24.403,421.463,169.449,35.860,156.754
C08590=1042.307,-24.154,421.450,169.451,35.861,156.755
C08591=1042.313,-23.904,421.436,169.453,35.862,156.755
C08592=1042.320,-23.654,421.422,169.455,35.862,156.755
C08593=1042.326,-23.404,421.409,169.457,35.864,156.755
C08594=1042.332,-23.156,421.394,169.459,35.864,156.755
C08595=1042.338,-22.906,421.381,169.461,35.865,156.755
C08596=1042.345,-22.656,421.367,169.463,35.866,156.755
C08597=1042.351,-22.407,421.353,169.465,35.867,156.756
C08598=1042.358,-22.157,421.339,169.467,35.868,156.756
C08599=1042.363,-21.908,421.325,169.469,35.868,156.756
C08600=1042.370,-21.658,421.311,169.471,35.869,156.756
C08601=1042.376,-21.409,421.298,169.473,35.870,156.756
C08602=1042.383,-21.159,421.283,169.476,35.871,156.756
C08603=1042.389,-20.910,421.270,169.478,35.872,156.756
C08604=1042.395,-20.659,421.256,169.480,35.873,156.757
C08605=1042.401,-20.411,421.242,169.482,35.874,156.757
C08606=1042.408,-20.161,421.228,169.484,35.874,156.757
C08607=1042.414,-19.911,421.214,169.486,35.875,156.757
C08608=1042.421,-19.629,421.198,169.489,35.876,156.757
C08609=1042.428,-19.348,421.182,169.491,35.877,156.757
C08610=1042.435,-19.066,421.167,169.493,35.878,156.757
C08611=1042.443,-18.784,421.151,169.496,35.879,156.758
C08612=1042.449,-18.535,421.138,169.498,35.880,156.758
C08613=1042.456,-18.285,421.123,169.500,35.881,156.758
C08614=1042.462,-18.036,421.109,169.502,35.882,156.758
C08615=1042.468,-17.786,421.095,169.504,35.882,156.758
C08616=1042.474,-17.537,421.081,169.507,35.884,156.758
C08617=1042.480,-17.287,421.067,169.509,35.884,156.758
C08618=1042.487,-17.038,421.053,169.511,35.885,156.759
C08619=1042.494,-16.788,421.039,169.513,35.886,156.759
C08620=1042.500,-16.538,421.024,169.515,35.887,156.759
C08621=1042.506,-16.289,421.011,169.517,35.888,156.759
C08622=1042.512,-16.039,420.997,169.519,35.888,156.759
C08623=1042.519,-15.790,420.983,169.521,35.890,156.759
C08624=1042.525,-15.540,420.969,169.523,35.890,156.759
C08625=1042.532,-15.291,420.955,169.525,35.891,156.760
C08626=1042.538,-15.041,420.941,169.527,35.892,156.760
C08627=1042.545,-14.792,420.926,169.529,35.893,156.760
C08628=1042.550,-14.542,420.912,169.531,35.894,156.760
C08629=1042.557,-14.292,420.897,169.533,35.895,156.760
C08630=1042.563,-14.043,420.884,169.535,35.896,156.760
C08631=1042.569,-13.793,420.869,169.538,35.897,156.761
C08632=1042.575,-13.545,420.855,169.540,35.898,156.761
C08633=1042.582,-13.295,420.841,169.542,35.899,156.761
C08634=1042.588,-13.045,420.826,169.544,35.900,156.761
C08635=1042.594,-12.795,420.812,169.546,35.900,156.761
C08636=1042.601,-12.546,420.798,169.548,35.902,156.761
C08637=1042.607,-12.297,420.783,169.549,35.902,156.761
C08638=1042.613,-12.047,420.769,169.551,35.903,156.762
C08639=1042.620,-11.797,420.755,169.553,35.904,156.762
C08640=1042.626,-11.548,420.740,169.555,35.905,156.762
C08641=1042.632,-11.298,420.726,169.557,35.906,156.762
C08642=1042.638,-11.050,420.712,169.559,35.907,156.762
C08643=1042.644,-10.799,420.698,169.562,35.908,156.762
C08644=1042.651,-10.550,420.683,169.564,35.909,156.763
C08645=1042.657,-10.301,420.669,169.566,35.910,156.763
C08646=1042.663,-10.051,420.654,169.568,35.911,156.763
C08647=1042.670,-9.801,420.639,169.570,35.912,156.763
C08648=1042.676,-9.552,420.625,169.572,35.913,156.763
C08649=1042.683,-9.303,420.611,169.574,35.914,156.763
C08650=1042.689,-9.052,420.596,169.576,35.915,156.763
C08651=1042.695,-8.804,420.582,169.578,35.915,156.764
C08652=1042.701,-8.554,420.567,169.580,35.917,156.764
C08653=1042.708,-8.304,420.553,169.582,35.917,156.764
C08654=1042.713,-8.055,420.539,169.584,35.919,156.764
C08655=1042.720,-7.806,420.524,169.586,35.919,156.764
C08656=1042.727,-7.556,420.509,169.589,35.921,156.764
C08657=1042.733,-7.307,420.495,169.591,35.921,156.765
C08658=1042.739,-7.057,420.481,169.593,35.923,156.765
C08659=1042.746,-6.807,420.466,169.595,35.923,156.765
C08660=1042.752,-6.558,420.451,169.597,35.924,156.765
C08661=1042.758,-6.309,420.437,169.599,35.925,156.765
C08662=1042.765,-6.059,420.423,169.600,35.926,156.765
C08663=1042.771,-5.809,420.408,169.602,35.927,156.766
C08664=1042.777,-5.560,420.393,169.604,35.928,156.766
C08665=1042.784,-5.311,420.379,169.606,35.929,156.766
C08666=1042.790,-5.061,420.364,169.608,35.930,156.766
C08667=1042.797,-4.811,420.349,169.610,35.930,156.766
C08668=1042.802,-4.562,420.335,169.612,35.932,156.766
C08669=1042.809,-4.313,420.321,169.615,35.932,156.766
C08670=1042.816,-4.063,420.306,169.617,35.934,156.767
C08671=1042.822,-3.813,420.291,169.619,35.934,156.767
C08672=1042.829,-3.530,420.275,169.621,35.936,156.767
C08673=1042.837,-3.247,420.258,169.623,35.937,156.767
C08674=1042.844,-2.963,420.241,169.625,35.938,156.767
C08675=1042.850,-2.680,420.224,169.628,35.939,156.768
C08676=1042.857,-2.431,420.209,169.630,35.940,156.768
C08677=1042.863,-2.181,420.194,169.631,35.942,156.768
C08678=1042.869,-1.932,420.179,169.633,35.942,156.768
C08679=1042.875,-1.682,420.164,169.635,35.944,156.768
C08680=1042.882,-1.433,420.149,169.638,35.945,156.769
C08681=1042.888,-1.183,420.134,169.640,35.945,156.769
C08682=1042.894,-0.934,420.120,169.642,35.947,156.769
C08683=1042.900,-0.684,420.105,169.644,35.947,156.769
C08684=1042.907,-0.435,420.090,169.646,35.949,156.769
C08685=1042.913,-0.185,420.075,169.648,35.950,156.769
C08686=1042.919,0.064,420.060,169.649,35.951,156.770
C08687=1042.925,0.314,420.045,169.651,35.952,156.770
C08688=1042.932,0.563,420.030,169.653,35.953,156.770
C08689=1042.938,0.813,420.015,169.655,35.954,156.770
C08690=1042.944,1.063,420.001,169.658,35.955,156.770
C08691=1042.950,1.311,419.986,169.660,35.957,156.771
C08692=1042.957,1.561,419.971,169.662,35.957,156.771
C08693=1042.962,1.811,419.955,169.664,35.959,156.771
C08694=1042.969,2.061,419.941,169.666,35.959,156.771
C08695=1042.975,2.310,419.925,169.667,35.960,156.771
C08696=1042.981,2.559,419.910,169.669,35.962,156.771
C08697=1042.987,2.808,419.895,169.671,35.962,156.772
C08698=1042.994,3.058,419.880,169.673,35.964,156.772
C08699=1043.000,3.308,419.865,169.675,35.965,156.772
C08700=1043.007,3.557,419.850,169.677,35.966,156.772
C08701=1043.013,3.806,419.835,169.680,35.967,156.772
C08702=1043.019,4.055,419.820,169.682,35.968,156.772
C08703=1043.025,4.305,419.805,169.683,35.969,156.773
C08704=1043.032,4.555,419.790,169.685,35.970,156.773
C08705=1043.038,4.804,419.775,169.687,35.971,156.773
C08706=1043.045,5.054,419.760,169.689,35.972,156.773
C08707=1043.051,5.303,419.744,169.691,35.973,156.773
C08708=1043.057,5.553,419.729,169.693,35.974,156.774
C08709=1043.063,5.803,419.714,169.695,35.975,156.774
C08710=1043.069,6.052,419.700,169.697,35.976,156.774
C08711=1043.076,6.301,419.684,169.698,35.977,156.774
C08712=1043.082,6.550,419.669,169.701,35.979,156.774
C08713=1043.089,6.800,419.654,169.703,35.979,156.775
C08714=1043.095,7.050,419.639,169.705,35.981,156.775
C08715=1043.102,7.299,419.624,169.707,35.982,156.775
C08716=1043.108,7.548,419.609,169.709,35.983,156.775
C08717=1043.114,7.798,419.593,169.711,35.984,156.775
C08718=1043.120,8.047,419.577,169.713,35.985,156.775
C08719=1043.127,8.297,419.562,169.714,35.986,156.776
C08720=1043.133,8.547,419.548,169.716,35.987,156.776
C08721=1043.140,8.796,419.532,169.718,35.988,156.776
C08722=1043.146,9.045,419.517,169.720,35.989,156.776
C08723=1043.153,9.295,419.502,169.723,35.990,156.776
C08724=1043.159,9.544,419.486,169.725,35.991,156.777
C08725=1043.165,9.793,419.472,169.727,35.992,156.777
C08726=1043.171,10.043,419.456,169.728,35.993,156.777
C08727=1043.177,10.292,419.441,169.730,35.994,156.777
C08728=1043.184,10.542,419.426,169.732,35.996,156.777
C08729=1043.190,10.791,419.411,169.734,35.996,156.777
C08730=1043.197,11.040,419.395,169.736,35.998,156.778
C08731=1043.203,11.290,419.380,169.738,35.998,156.778
C08732=1043.210,11.539,419.364,169.740,36.000,156.778
C08733=1043.216,11.789,419.349,169.741,36.001,156.778
C08734=1043.222,12.039,419.334,169.744,36.001,156.778
C08735=1043.229,12.288,419.318,169.746,36.003,156.779
C08736=1043.236,12.573,419.301,169.748,36.004,156.779
C08737=1043.243,12.859,419.284,169.750,36.005,156.779
C08738=1043.251,13.144,419.266,169.753,36.006,156.779
C08739=1043.258,13.429,419.248,169.755,36.007,156.779
C08740=1043.265,13.678,419.233,169.757,36.009,156.780
C08741=1043.271,13.928,419.218,169.758,36.009,156.780
C08742=1043.277,14.177,419.201,169.760,36.011,156.780
C08743=1043.284,14.427,419.186,169.762,36.012,156.780
C08744=1043.291,14.676,419.171,169.765,36.013,156.780
C08745=1043.296,14.926,419.155,169.767,36.014,156.780
C08746=1043.303,15.175,419.140,169.769,36.015,156.781
C08747=1043.308,15.425,419.124,169.770,36.016,156.781
C08748=1043.315,15.674,419.108,169.772,36.018,156.781
C08749=1043.322,15.924,419.093,169.774,36.018,156.781
C08750=1043.328,16.173,419.077,169.776,36.020,156.781
C08751=1043.334,16.422,419.061,169.778,36.021,156.782
C08752=1043.340,16.672,419.046,169.779,36.022,156.782
C08753=1043.347,16.921,419.030,169.781,36.023,156.782
C08754=1043.354,17.171,419.014,169.784,36.024,156.782
C08755=1043.359,17.421,418.999,169.786,36.025,156.782
C08756=1043.366,17.670,418.983,169.788,36.027,156.783
C08757=1043.372,17.920,418.968,169.790,36.027,156.783
C08758=1043.378,18.169,418.952,169.791,36.029,156.783
C08759=1043.385,18.418,418.936,169.793,36.030,156.783
C08760=1043.391,18.668,418.921,169.795,36.031,156.784
C08761=1043.398,18.917,418.905,169.797,36.032,156.784
C08762=1043.403,19.166,418.889,169.799,36.033,156.784
C08763=1043.410,19.416,418.874,169.801,36.034,156.784
C08764=1043.417,19.665,418.858,169.803,36.035,156.784
C08765=1043.422,19.914,418.842,169.805,36.036,156.784
C08766=1043.430,20.164,418.826,169.807,36.038,156.785
C08767=1043.435,20.414,418.810,169.809,36.039,156.785
C08768=1043.442,20.663,418.795,169.810,36.040,156.785
C08769=1043.448,20.912,418.778,169.812,36.041,156.785
C08770=1043.454,21.162,418.762,169.814,36.042,156.785
C08771=1043.460,21.411,418.747,169.816,36.043,156.786
C08772=1043.466,21.661,418.731,169.818,36.045,156.786
C08773=1043.473,21.910,418.715,169.820,36.046,156.786
C08774=1043.479,22.159,418.699,169.822,36.047,156.786
C08775=1043.486,22.408,418.683,169.824,36.048,156.786
C08776=1043.492,22.659,418.667,169.826,36.049,156.787
C08777=1043.499,22.908,418.652,169.828,36.051,156.787
C08778=1043.505,23.157,418.636,169.829,36.052,156.787
C08779=1043.511,23.406,418.620,169.831,36.053,156.787
C08780=1043.517,23.655,418.604,169.833,36.054,156.787
C08781=1043.523,23.905,418.587,169.835,36.055,156.788
C08782=1043.530,24.154,418.572,169.837,36.056,156.788
C08783=1043.536,24.405,418.556,169.839,36.058,156.788
C08784=1043.543,24.654,418.540,169.841,36.059,156.788
C08785=1043.549,24.903,418.524,169.843,36.060,156.788
C08786=1043.555,25.152,418.508,169.845,36.061,156.789
C08787=1043.561,25.401,418.492,169.846,36.062,156.789
C08788=1043.567,25.651,418.476,169.848,36.063,156.789
C08789=1043.575,25.900,418.460,169.850,36.064,156.789
C08790=1043.581,26.150,418.443,169.852,36.065,156.790
C08791=1043.587,26.399,418.428,169.854,36.067,156.790
C08792=1043.593,26.649,418.412,169.856,36.068,156.790
C08793=1043.599,26.898,418.396,169.858,36.069,156.790
C08794=1043.606,27.148,418.380,169.860,36.071,156.790
C08795=1043.612,27.397,418.364,169.862,36.071,156.791
C08796=1043.619,27.646,418.348,169.863,36.072,156.791
C08797=1043.625,27.896,418.332,169.865,36.074,156.791
C08798=1043.631,28.145,418.315,169.867,36.075,156.791
C08799=1043.638,28.395,418.299,169.869,36.076,156.791
C08800=1043.645,28.681,418.280,169.871,36.078,156.792
C08801=1043.652,28.967,418.262,169.874,36.079,156.792
C08802=1043.659,29.254,418.244,169.876,36.080,156.792
C08803=1043.667,29.541,418.225,169.878,36.081,156.792
C08804=1043.672,29.790,418.209,169.880,36.083,156.793
C08805=1043.679,30.040,418.192,169.881,36.084,156.793
C08806=1043.685,30.289,418.176,169.883,36.085,156.793
C08807=1043.691,30.539,418.160,169.885,36.087,156.793
C08808=1043.698,30.788,418.144,169.887,36.088,156.794
C08809=1043.704,31.037,418.127,169.889,36.089,156.794
C08810=1043.710,31.286,418.110,169.891,36.090,156.794
C08811=1043.716,31.536,418.094,169.893,36.092,156.794
C08812=1043.722,31.785,418.078,169.895,36.092,156.794
C08813=1043.730,32.035,418.062,169.896,36.094,156.795
C08814=1043.736,32.284,418.046,169.898,36.095,156.795
C08815=1043.742,32.534,418.029,169.900,36.096,156.795
C08816=1043.747,32.783,418.013,169.902,36.097,156.795
C08817=1043.754,33.032,417.996,169.903,36.099,156.795
C08818=1043.761,33.281,417.980,169.906,36.100,156.796
C08819=1043.767,33.531,417.964,169.908,36.101,156.796
C08820=1043.773,33.780,417.948,169.910,36.103,156.796
C08821=1043.779,34.030,417.931,169.911,36.103,156.796
C08822=1043.786,34.279,417.914,169.913,36.105,156.796
C08823=1043.792,34.528,417.898,169.915,36.106,156.797
C08824=1043.799,34.778,417.882,169.917,36.107,156.797
C08825=1043.805,35.027,417.865,169.918,36.108,156.797
C08826=1043.811,35.277,417.849,169.920,36.110,156.797
C08827=1043.818,35.526,417.832,169.923,36.111,156.798
C08828=1043.824,35.775,417.816,169.925,36.112,156.798
C08829=1043.830,36.025,417.799,169.926,36.113,156.798
C08830=1043.837,36.275,417.783,169.928,36.114,156.798
C08831=1043.843,36.523,417.766,169.930,36.115,156.798
C08832=1043.849,36.773,417.750,169.932,36.117,156.799
C08833=1043.856,37.023,417.733,169.933,36.118,156.799
C08834=1043.862,37.271,417.716,169.935,36.119,156.799
C08835=1043.868,37.521,417.700,169.938,36.121,156.799
C08836=1043.874,37.771,417.684,169.940,36.122,156.800
C08837=1043.880,38.020,417.667,169.941,36.123,156.800
C08838=1043.887,38.269,417.650,169.943,36.124,156.800
C08839=1043.893,38.519,417.634,169.945,36.126,156.800
C08840=1043.899,38.768,417.617,169.946,36.127,156.801
C08841=1043.905,39.017,417.600,169.948,36.128,156.801
C08842=1043.912,39.267,417.584,169.950,36.129,156.801
C08843=1043.918,39.516,417.567,169.953,36.131,156.801
C08844=1043.924,39.765,417.551,169.954,36.132,156.801
C08845=1043.931,40.015,417.533,169.956,36.133,156.802
C08846=1043.937,40.264,417.517,169.958,36.134,156.802
C08847=1043.944,40.514,417.500,169.959,36.135,156.802
C08848=1043.950,40.763,417.483,169.961,36.137,156.802
C08849=1043.956,41.012,417.467,169.963,36.138,156.802
C08850=1043.963,41.261,417.450,169.965,36.139,156.803
C08851=1043.969,41.511,417.434,169.966,36.140,156.803
C08852=1043.974,41.760,417.416,169.969,36.142,156.803
C08853=1043.981,42.010,417.399,169.971,36.143,156.803
C08854=1043.987,42.259,417.382,169.973,36.144,156.804
C08855=1043.993,42.509,417.366,169.974,36.145,156.804
C08856=1043.999,42.758,417.350,169.976,36.147,156.804
C08857=1044.006,43.007,417.333,169.978,36.148,156.804
C08858=1044.012,43.256,417.315,169.979,36.149,156.805
C08859=1044.018,43.506,417.299,169.981,36.151,156.805
C08860=1044.025,43.755,417.282,169.984,36.152,156.805
C08861=1044.031,44.005,417.265,169.986,36.153,156.805
C08862=1044.037,44.253,417.248,169.987,36.154,156.805
C08863=1044.043,44.503,417.231,169.989,36.156,156.806
C08864=1044.050,44.789,417.211,169.991,36.158,156.806
C08865=1044.057,45.076,417.192,169.993,36.159,156.806
C08866=1044.064,45.363,417.172,169.995,36.161,156.807
C08867=1044.071,45.649,417.152,169.998,36.162,156.807
C08868=1044.077,45.898,417.135,169.999,36.163,156.807
C08869=1044.084,46.148,417.119,170.001,36.165,156.807
C08870=1044.089,46.397,417.101,170.003,36.166,156.808
C08871=1044.096,46.647,417.085,170.004,36.167,156.808
C08872=1044.102,46.896,417.068,170.006,36.169,156.808
C08873=1044.108,47.145,417.050,170.008,36.170,156.808
C08874=1044.114,47.395,417.033,170.010,36.172,156.809
C08875=1044.121,47.644,417.017,170.012,36.173,156.809
C08876=1044.127,47.893,416.999,170.014,36.174,156.809
C08877=1044.133,48.142,416.982,170.016,36.175,156.809
C08878=1044.140,48.392,416.965,170.017,36.177,156.810
C08879=1044.145,48.641,416.947,170.019,36.178,156.810
C08880=1044.152,48.891,416.930,170.021,36.179,156.810
C08881=1044.158,49.140,416.914,170.022,36.180,156.810
C08882=1044.164,49.390,416.896,170.024,36.182,156.810
C08883=1044.170,49.638,416.879,170.027,36.183,156.811
C08884=1044.177,49.888,416.862,170.028,36.184,156.811
C08885=1044.182,50.137,416.845,170.030,36.186,156.811
C08886=1044.189,50.387,416.827,170.032,36.187,156.811
C08887=1044.195,50.636,416.810,170.033,36.189,156.812
C08888=1044.202,50.885,416.792,170.035,36.190,156.812
C08889=1044.208,51.135,416.776,170.037,36.191,156.812
C08890=1044.214,51.384,416.758,170.040,36.193,156.812
C08891=1044.220,51.633,416.741,170.041,36.194,156.813
C08892=1044.227,51.883,416.724,170.043,36.195,156.813
C08893=1044.232,52.132,416.706,170.045,36.196,156.813
C08894=1044.239,52.382,416.690,170.046,36.198,156.813
C08895=1044.245,52.630,416.673,170.048,36.199,156.814
C08896=1044.251,52.880,416.655,170.050,36.200,156.814
C08897=1044.257,53.129,416.638,170.051,36.201,156.814
C08898=1044.264,53.378,416.621,170.054,36.203,156.814
C08899=1044.270,53.627,416.603,170.056,36.204,156.814
C08900=1044.277,53.877,416.586,170.058,36.205,156.815
C08901=1044.282,54.126,416.569,170.059,36.207,156.815
C08902=1044.289,54.376,416.551,170.061,36.208,156.815
C08903=1044.296,54.625,416.534,170.063,36.209,156.815
C08904=1044.301,54.874,416.517,170.064,36.210,156.816
C08905=1044.308,55.124,416.499,170.066,36.212,156.816
C08906=1044.314,55.373,416.482,170.069,36.213,156.816
C08907=1044.320,55.622,416.464,170.070,36.215,156.816
C08908=1044.327,55.872,416.447,170.072,36.216,156.817
C08909=1044.333,56.121,416.429,170.074,36.217,156.817
C08910=1044.340,56.370,416.412,170.075,36.219,156.817
C08911=1044.346,56.619,416.395,170.077,36.220,156.817
C08912=1044.352,56.869,416.378,170.079,36.221,156.818
C08913=1044.359,57.119,416.361,170.082,36.222,156.818
C08914=1044.364,57.368,416.343,170.083,36.224,156.818
C08915=1044.371,57.617,416.326,170.085,36.225,156.818
C08916=1044.377,57.866,416.309,170.087,36.226,156.819
C08917=1044.383,58.116,416.291,170.088,36.227,156.819
C08918=1044.390,58.365,416.273,170.090,36.229,156.819
C08919=1044.396,58.614,416.256,170.092,36.230,156.819
C08920=1044.403,58.863,416.239,170.093,36.231,156.819
C08921=1044.409,59.113,416.221,170.096,36.233,156.820
C08922=1044.415,59.362,416.204,170.098,36.234,156.820
C08923=1044.422,59.611,416.186,170.100,36.235,156.820
C08924=1044.428,59.861,416.168,170.101,36.236,156.820
C08925=1044.434,60.109,416.151,170.103,36.238,156.821
C08926=1044.441,60.359,416.133,170.105,36.239,156.821
C08927=1044.447,60.608,416.115,170.106,36.240,156.821
C08928=1044.454,60.894,416.095,170.108,36.241,156.821
C08929=1044.462,61.181,416.075,170.111,36.243,156.822
C08930=1044.469,61.467,416.055,170.113,36.245,156.822
C08931=1044.476,61.754,416.035,170.115,36.246,156.822
C08932=1044.483,62.002,416.018,170.117,36.247,156.822
C08933=1044.489,62.252,416.000,170.119,36.248,156.823
C08934=1044.496,62.501,415.983,170.120,36.250,156.823
C08935=1044.503,62.751,415.965,170.122,36.251,156.823
C08936=1044.508,62.999,415.947,170.125,36.252,156.823
C08937=1044.515,63.249,415.930,170.126,36.253,156.824
C08938=1044.521,63.498,415.912,170.128,36.255,156.824
C08939=1044.528,63.748,415.894,170.130,36.256,156.824
C08940=1044.534,63.997,415.877,170.131,36.257,156.824
C08941=1044.541,64.246,415.859,170.133,36.259,156.824
C08942=1044.547,64.495,415.841,170.135,36.260,156.825
C08943=1044.553,64.745,415.823,170.136,36.261,156.825
C08944=1044.559,64.994,415.806,170.139,36.262,156.825
C08945=1044.566,65.244,415.788,170.141,36.264,156.825
C08946=1044.572,65.493,415.769,170.143,36.266,156.826
C08947=1044.578,65.742,415.752,170.144,36.267,156.826
C08948=1044.584,65.991,415.734,170.146,36.268,156.826
C08949=1044.590,66.241,415.716,170.148,36.269,156.826
C08950=1044.596,66.489,415.698,170.149,36.271,156.827
C08951=1044.603,66.739,415.681,170.152,36.272,156.827
C08952=1044.609,66.989,415.663,170.154,36.273,156.827
C08953=1044.616,67.238,415.644,170.155,36.274,156.827
C08954=1044.622,67.486,415.627,170.157,36.276,156.828
C08955=1044.628,67.736,415.609,170.159,36.278,156.828
C08956=1044.634,67.985,415.591,170.160,36.279,156.828
C08957=1044.641,68.235,415.573,170.162,36.280,156.828
C08958=1044.646,68.484,415.555,170.165,36.281,156.829
C08959=1044.653,68.733,415.537,170.166,36.283,156.829
C08960=1044.659,68.983,415.519,170.168,36.284,156.829
C08961=1044.666,69.232,415.501,170.170,36.285,156.829
C08962=1044.672,69.482,415.483,170.171,36.286,156.830
C08963=1044.678,69.730,415.466,170.173,36.288,156.830
C08964=1044.685,69.979,415.447,170.175,36.290,156.830
C08965=1044.691,70.229,415.429,170.177,36.291,156.830
C08966=1044.697,70.479,415.411,170.179,36.292,156.831
C08967=1044.703,70.727,415.393,170.181,36.293,156.831
C08968=1044.709,70.977,415.375,170.182,36.295,156.831
C08969=1044.715,71.226,415.356,170.184,36.296,156.832
C08970=1044.721,71.476,415.338,170.186,36.298,156.832
C08971=1044.728,71.724,415.321,170.187,36.299,156.832
C08972=1044.734,71.974,415.303,170.190,36.300,156.832
C08973=1044.740,72.223,415.284,170.192,36.301,156.832
C08974=1044.747,72.473,415.266,170.193,36.303,156.833
C08975=1044.753,72.722,415.248,170.195,36.305,156.833
C08976=1044.759,72.971,415.230,170.197,36.306,156.833
C08977=1044.765,73.220,415.211,170.198,36.307,156.834
C08978=1044.771,73.470,415.193,170.200,36.308,156.834
C08979=1044.778,73.719,415.175,170.203,36.310,156.834
C08980=1044.784,73.969,415.157,170.204,36.312,156.834
C08981=1044.790,74.218,415.138,170.206,36.313,156.835
C08982=1044.796,74.467,415.121,170.208,36.314,156.835
C08983=1044.802,74.716,415.102,170.209,36.315,156.835
C08984=1044.809,74.965,415.084,170.211,36.317,156.835
C08985=1044.815,75.214,415.066,170.213,36.318,156.836
C08986=1044.822,75.463,415.047,170.215,36.320,156.836
C08987=1044.828,75.713,415.029,170.217,36.321,156.836
C08988=1044.834,75.962,415.011,170.219,36.322,156.836
C08989=1044.840,76.211,414.992,170.220,36.324,156.837
C08990=1044.846,76.460,414.975,170.222,36.325,156.837
C08991=1044.853,76.710,414.956,170.224,36.326,156.837
C08992=1044.860,76.996,414.934,170.226,36.328,156.837
C08993=1044.867,77.282,414.914,170.229,36.329,156.838
C08994=1044.874,77.568,414.893,170.230,36.331,156.838
C08995=1044.881,77.853,414.872,170.232,36.332,156.838
C08996=1044.888,78.103,414.853,170.234,36.334,156.839
C08997=1044.894,78.352,414.835,170.236,36.335,156.839
C08998=1044.900,78.601,414.817,170.237,36.337,156.839
C08999=1044.906,78.851,414.798,170.240,36.338,156.839
C09000=1044.912,79.100,414.779,170.242,36.340,156.840
C09001=1044.918,79.350,414.761,170.243,36.341,156.840
C09002=1044.924,79.598,414.743,170.245,36.342,156.840
C09003=1044.931,79.847,414.724,170.247,36.344,156.840
C09004=1044.936,80.097,414.705,170.248,36.346,156.841
C09005=1044.943,80.346,414.686,170.250,36.347,156.841
C09006=1044.949,80.596,414.668,170.253,36.348,156.841
C09007=1044.955,80.845,414.650,170.254,36.349,156.841
C09008=1044.962,81.094,414.631,170.256,36.351,156.842
C09009=1044.967,81.343,414.612,170.258,36.352,156.842
C09010=1044.974,81.592,414.593,170.259,36.354,156.842
C09011=1044.979,81.841,414.575,170.261,36.355,156.842
C09012=1044.986,82.091,414.557,170.264,36.357,156.843
C09013=1044.992,82.340,414.538,170.265,36.358,156.843
C09014=1044.998,82.589,414.519,170.267,36.359,156.843
C09015=1045.004,82.838,414.500,170.269,36.361,156.844
C09016=1045.011,83.087,414.482,170.270,36.363,156.844
C09017=1045.017,83.337,414.464,170.272,36.364,156.844
C09018=1045.023,83.586,414.445,170.274,36.365,156.844
C09019=1045.029,83.836,414.426,170.276,36.366,156.845
C09020=1045.035,84.085,414.407,170.278,36.368,156.845
C09021=1045.042,84.334,414.388,170.280,36.369,156.845
C09022=1045.048,84.583,414.370,170.281,36.371,156.845
C09023=1045.054,84.832,414.351,170.283,36.372,156.846
C09024=1045.060,85.082,414.332,170.285,36.374,156.846
C09025=1045.067,85.331,414.313,170.287,36.375,156.846
C09026=1045.073,85.580,414.295,170.289,36.376,156.846
C09027=1045.080,85.829,414.276,170.291,36.378,156.847
C09028=1045.085,86.078,414.257,170.292,36.379,156.847
C09029=1045.092,86.328,414.238,170.294,36.381,156.847
C09030=1045.098,86.577,414.220,170.296,36.382,156.848
C09031=1045.104,86.826,414.201,170.297,36.383,156.848
C09032=1045.110,87.076,414.182,170.300,36.384,156.848
C09033=1045.116,87.325,414.164,170.302,36.386,156.848
C09034=1045.123,87.574,414.145,170.303,36.388,156.849
C09035=1045.129,87.823,414.126,170.305,36.389,156.849
C09036=1045.135,88.073,414.107,170.307,36.390,156.849
C09037=1045.141,88.322,414.088,170.308,36.391,156.849
C09038=1045.148,88.571,414.070,170.310,36.393,156.850
C09039=1045.155,88.819,414.050,170.313,36.395,156.850
C09040=1045.160,89.069,414.031,170.314,36.396,156.850
C09041=1045.167,89.318,414.013,170.316,36.397,156.850
C09042=1045.173,89.567,413.994,170.318,36.398,156.851
C09043=1045.179,89.816,413.975,170.319,36.400,156.851
C09044=1045.185,90.066,413.956,170.321,36.401,156.851
C09045=1045.192,90.315,413.937,170.324,36.403,156.851
C09046=1045.198,90.564,413.919,170.325,36.404,156.852
C09047=1045.204,90.813,413.899,170.327,36.406,156.852
C09048=1045.210,91.062,413.881,170.329,36.407,156.852
C09049=1045.216,91.312,413.862,170.330,36.408,156.853
C09050=1045.223,91.560,413.842,170.332,36.410,156.853
C09051=1045.228,91.810,413.823,170.334,36.411,156.853
C09052=1045.234,92.059,413.804,170.336,36.413,156.853
C09053=1045.240,92.308,413.785,170.338,36.415,156.854
C09054=1045.247,92.558,413.765,170.340,36.416,156.854
C09055=1045.253,92.807,413.746,170.341,36.417,156.854
C09056=1045.260,93.093,413.725,170.343,36.419,156.855
C09057=1045.267,93.379,413.703,170.346,36.421,156.855
C09058=1045.274,93.665,413.681,170.348,36.422,156.855
C09059=1045.281,93.951,413.659,170.350,36.424,156.855
C09060=1045.288,94.200,413.639,170.352,36.425,156.856
C09061=1045.293,94.449,413.620,170.353,36.426,156.856
C09062=1045.300,94.698,413.601,170.355,36.428,156.856
C09063=1045.305,94.948,413.582,170.357,36.430,156.857
C09064=1045.312,95.196,413.563,170.359,36.431,156.857
C09065=1045.318,95.446,413.544,170.361,36.433,156.857
C09066=1045.324,95.695,413.525,170.363,36.434,156.857
C09067=1045.331,95.944,413.505,170.365,36.435,156.858
C09068=1045.337,96.193,413.486,170.366,36.437,156.858
C09069=1045.343,96.443,413.467,170.368,36.438,156.858
C09070=1045.349,96.692,413.447,170.371,36.440,156.858
C09071=1045.355,96.941,413.428,170.372,36.441,156.859
C09072=1045.361,97.190,413.409,170.374,36.443,156.859
C09073=1045.368,97.439,413.389,170.376,36.444,156.859
C09074=1045.373,97.688,413.370,170.377,36.445,156.860
C09075=1045.381,97.938,413.351,170.379,36.447,156.860
C09076=1045.386,98.153,413.334,170.381,36.448,156.860
C09077=1045.391,98.367,413.317,170.383,36.450,156.860
C09078=1045.396,98.582,413.301,170.384,36.451,156.861
C09079=1045.401,98.797,413.285,170.386,36.452,156.861
C09080=1045.407,99.011,413.268,170.387,36.453,156.861
C09081=1045.412,99.227,413.251,170.389,36.454,156.861
C09082=1045.418,99.441,413.235,170.390,36.455,156.861
C09083=1045.423,99.655,413.218,170.392,36.456,156.862
C09084=1045.429,99.905,413.198,170.394,36.458,156.862
C09085=1045.436,100.153,413.179,170.396,36.460,156.862
C09086=1045.442,100.403,413.159,170.398,36.461,156.863
C09087=1045.448,100.653,413.140,170.399,36.462,156.863
C09088=1045.454,100.901,413.121,170.401,36.464,156.863
C09089=1045.460,101.150,413.101,170.403,36.465,156.863
C09090=1045.466,101.400,413.082,170.405,36.467,156.864
C09091=1045.472,101.648,413.062,170.407,36.468,156.864
C09092=1045.478,101.899,413.042,170.409,36.470,156.864
C09093=1045.485,102.147,413.023,170.411,36.471,156.865
C09094=1045.491,102.397,413.003,170.412,36.473,156.865
C09095=1045.497,102.645,412.984,170.415,36.474,156.865
C09096=1045.503,102.895,412.964,170.417,36.476,156.865
C09097=1045.509,103.144,412.944,170.418,36.477,156.866
C09098=1045.515,103.394,412.925,170.420,36.479,156.866
C09099=1045.522,103.642,412.905,170.422,36.480,156.866
C09100=1045.528,103.891,412.885,170.423,36.482,156.867
C09101=1045.533,104.140,412.866,170.426,36.483,156.867
C09102=1045.539,104.389,412.846,170.428,36.484,156.867
C09103=1045.546,104.639,412.827,170.429,36.486,156.867
C09104=1045.552,104.888,412.807,170.431,36.488,156.868
C09105=1045.558,105.137,412.787,170.433,36.489,156.868
